KUKA KRL program: sParallel2.src, sParallel2.dat

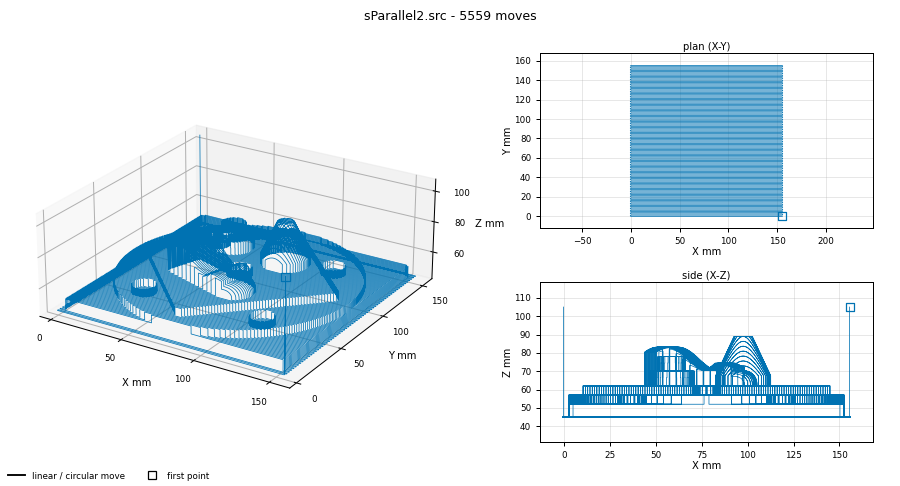
[picture p0: tool path of sParallel2.src, 5559 of 5560 moves have a stored position in this frame; points joined in program order, loops and branches not executed]
--- sParallel2.src ---
&ACCESS RVO
DEF sParallel2()
; Generated by AUTODESK Fusion 360 CAM 2.0.14793
; Creation date: Thursday, March 16, 2023 18:51:27
;FOLD sParallel2
; Start position (joint) = {A1 5,A2 -80,A3 100,A4 75,A5 -60,A6 -65}
; Tool Number            = 4
; Base Number            = 1
; Spindle Speed          = 5000 RPM
; Program file name      = sParallel2.src

PTP {A1 5,A2 -80,A3 100,A4 75,A5 -60,A6 -65,E1 0,E2 0,E3 0,E4 0,E5 0,E6 0}
LIN {X 155.508,Y -0.003,Z 105.000,A 180.000,B 0.000,C 180.000} C_DIS
LIN {X 155.508,Y -0.003,Z 47.000,A 180.000,B 0.000,C 180.000} C_DIS
; Plunge Move Starts
$VEL.CP=0.01
LIN {X 155.508,Y -0.003,Z 45.500,A 180.000,B 0.000,C 180.000} C_DIS
; Lead In Move Starts
LIN {X 155.361,Y -0.003,Z 45.146,A 180.000,B 0.000,C 180.000} C_DIS
LIN {X 155.008,Y -0.003,Z 45.000,A 180.000,B 0.000,C 180.000} C_DIS
; Cutting Move Starts
$VEL.CP=0.02
LIN {X -0.008,Y -0.003,Z 45.000,A 180.000,B 0.000,C 180.000} C_DIS
; Link Move Starts
LIN {X -0.118,Y -0.003,Z 45.026,A 180.000,B 0.000,C 180.000} C_DIS
LIN {X -0.228,Y -0.003,Z 45.051,A 180.000,B 0.000,C 180.000} C_DIS
LIN {X -0.230,Y -0.003,Z 45.051,A 180.000,B 0.000,C 180.000} C_DIS
LIN {X -0.771,Y 0.309,Z 45.051,A 180.000,B 0.000,C 180.000} C_DIS
LIN {X -0.771,Y 0.934,Z 45.051,A 180.000,B 0.000,C 180.000} C_DIS
LIN {X -0.230,Y 1.247,Z 45.051,A 180.000,B 0.000,C 180.000} C_DIS
LIN {X -0.120,Y 1.247,Z 45.026,A 180.000,B 0.000,C 180.000} C_DIS
LIN {X -0.010,Y 1.247,Z 45.000,A 180.000,B 0.000,C 180.000} C_DIS
; Cutting Move Starts
LIN {X 155.010,Y 1.247,Z 45.000,A 180.000,B 0.000,C 180.000} C_DIS
; Link Move Starts
LIN {X 155.120,Y 1.247,Z 45.026,A 180.000,B 0.000,C 180.000} C_DIS
LIN {X 155.230,Y 1.247,Z 45.051,A 180.000,B 0.000,C 180.000} C_DIS
LIN {X 155.771,Y 1.559,Z 45.051,A 180.000,B 0.000,C 180.000} C_DIS
LIN {X 155.771,Y 2.184,Z 45.051,A 180.000,B 0.000,C 180.000} C_DIS
LIN {X 155.230,Y 2.497,Z 45.051,A 180.000,B 0.000,C 180.000} C_DIS
LIN {X 155.120,Y 2.497,Z 45.026,A 180.000,B 0.000,C 180.000} C_DIS
LIN {X 155.010,Y 2.497,Z 45.000,A 180.000,B 0.000,C 180.000} C_DIS
; Cutting Move Starts
LIN {X -0.010,Y 2.497,Z 45.000,A 180.000,B 0.000,C 180.000} C_DIS
; Link Move Starts
LIN {X -0.120,Y 2.497,Z 45.026,A 180.000,B 0.000,C 180.000} C_DIS
LIN {X -0.230,Y 2.497,Z 45.051,A 180.000,B 0.000,C 180.000} C_DIS
LIN {X -0.771,Y 2.809,Z 45.051,A 180.000,B 0.000,C 180.000} C_DIS
LIN {X -0.771,Y 3.434,Z 45.051,A 180.000,B 0.000,C 180.000} C_DIS
LIN {X -0.230,Y 3.746,Z 45.051,A 180.000,B 0.000,C 180.000} C_DIS
LIN {X -0.120,Y 3.746,Z 45.026,A 180.000,B 0.000,C 180.000} C_DIS
LIN {X -0.010,Y 3.746,Z 45.000,A 180.000,B 0.000,C 180.000} C_DIS
; Cutting Move Starts
LIN {X 2.836,Y 3.746,Z 45.000,A 180.000,B 0.000,C 180.000} C_DIS
LIN {X 2.837,Y 3.746,Z 52.000,A 180.000,B 0.000,C 180.000} C_DIS
LIN {X 63.902,Y 3.746,Z 52.000,A 180.000,B 0.000,C 180.000} C_DIS
LIN {X 63.902,Y 3.746,Z 57.000,A 180.000,B 0.000,C 180.000} C_DIS
LIN {X 91.097,Y 3.746,Z 57.000,A 180.000,B 0.000,C 180.000} C_DIS
LIN {X 91.098,Y 3.746,Z 52.000,A 180.000,B 0.000,C 180.000} C_DIS
LIN {X 152.163,Y 3.746,Z 52.000,A 180.000,B 0.000,C 180.000} C_DIS
LIN {X 152.163,Y 3.746,Z 45.000,A 180.000,B 0.000,C 180.000} C_DIS
LIN {X 155.010,Y 3.746,Z 45.000,A 180.000,B 0.000,C 180.000} C_DIS
; Link Move Starts
LIN {X 155.120,Y 3.746,Z 45.026,A 180.000,B 0.000,C 180.000} C_DIS
LIN {X 155.230,Y 3.746,Z 45.051,A 180.000,B 0.000,C 180.000} C_DIS
LIN {X 155.771,Y 4.059,Z 45.051,A 180.000,B 0.000,C 180.000} C_DIS
LIN {X 155.771,Y 4.684,Z 45.051,A 180.000,B 0.000,C 180.000} C_DIS
LIN {X 155.230,Y 4.996,Z 45.051,A 180.000,B 0.000,C 180.000} C_DIS
LIN {X 155.120,Y 4.996,Z 45.026,A 180.000,B 0.000,C 180.000} C_DIS
LIN {X 155.010,Y 4.996,Z 45.000,A 180.000,B 0.000,C 180.000} C_DIS
; Cutting Move Starts
LIN {X 152.500,Y 4.996,Z 45.000,A 180.000,B 0.000,C 180.000} C_DIS
LIN {X 152.500,Y 4.996,Z 52.000,A 180.000,B 0.000,C 180.000} C_DIS
LIN {X 96.687,Y 4.996,Z 52.000,A 180.000,B 0.000,C 180.000} C_DIS
LIN {X 96.684,Y 4.996,Z 57.000,A 180.000,B 0.000,C 180.000} C_DIS
LIN {X 58.313,Y 4.996,Z 57.000,A 180.000,B 0.000,C 180.000} C_DIS
LIN {X 58.313,Y 4.996,Z 52.000,A 180.000,B 0.000,C 180.000} C_DIS
LIN {X 2.500,Y 4.996,Z 52.000,A 180.000,B 0.000,C 180.000} C_DIS
LIN {X 2.500,Y 4.996,Z 45.000,A 180.000,B 0.000,C 180.000} C_DIS
LIN {X -0.010,Y 4.996,Z 45.000,A 180.000,B 0.000,C 180.000} C_DIS
; Link Move Starts
LIN {X -0.120,Y 4.996,Z 45.026,A 180.000,B 0.000,C 180.000} C_DIS
LIN {X -0.230,Y 4.996,Z 45.051,A 180.000,B 0.000,C 180.000} C_DIS
LIN {X -0.771,Y 5.309,Z 45.051,A 180.000,B 0.000,C 180.000} C_DIS
LIN {X -0.771,Y 5.934,Z 45.051,A 180.000,B 0.000,C 180.000} C_DIS
LIN {X -0.230,Y 6.246,Z 45.051,A 180.000,B 0.000,C 180.000} C_DIS
LIN {X -0.120,Y 6.246,Z 45.026,A 180.000,B 0.000,C 180.000} C_DIS
LIN {X -0.010,Y 6.246,Z 45.000,A 180.000,B 0.000,C 180.000} C_DIS
; Cutting Move Starts
LIN {X 2.499,Y 6.246,Z 45.000,A 180.000,B 0.000,C 180.000} C_DIS
LIN {X 2.500,Y 6.246,Z 52.000,A 180.000,B 0.000,C 180.000} C_DIS
LIN {X 54.109,Y 6.246,Z 52.000,A 180.000,B 0.000,C 180.000} C_DIS
LIN {X 54.109,Y 6.246,Z 57.000,A 180.000,B 0.000,C 180.000} C_DIS
LIN {X 100.891,Y 6.246,Z 57.000,A 180.000,B 0.000,C 180.000} C_DIS
LIN {X 100.891,Y 6.246,Z 52.000,A 180.000,B 0.000,C 180.000} C_DIS
LIN {X 152.500,Y 6.246,Z 52.000,A 180.000,B 0.000,C 180.000} C_DIS
LIN {X 152.500,Y 6.246,Z 45.000,A 180.000,B 0.000,C 180.000} C_DIS
LIN {X 155.010,Y 6.246,Z 45.000,A 180.000,B 0.000,C 180.000} C_DIS
; Link Move Starts
LIN {X 155.120,Y 6.246,Z 45.026,A 180.000,B 0.000,C 180.000} C_DIS
LIN {X 155.230,Y 6.246,Z 45.051,A 180.000,B 0.000,C 180.000} C_DIS
LIN {X 155.771,Y 6.559,Z 45.051,A 180.000,B 0.000,C 180.000} C_DIS
LIN {X 155.771,Y 7.184,Z 45.051,A 180.000,B 0.000,C 180.000} C_DIS
LIN {X 155.230,Y 7.496,Z 45.051,A 180.000,B 0.000,C 180.000} C_DIS
LIN {X 155.120,Y 7.496,Z 45.026,A 180.000,B 0.000,C 180.000} C_DIS
LIN {X 155.010,Y 7.496,Z 45.000,A 180.000,B 0.000,C 180.000} C_DIS
; Cutting Move Starts
LIN {X 152.500,Y 7.496,Z 45.000,A 180.000,B 0.000,C 180.000} C_DIS
LIN {X 152.500,Y 7.496,Z 52.000,A 180.000,B 0.000,C 180.000} C_DIS
LIN {X 104.403,Y 7.496,Z 52.000,A 180.000,B 0.000,C 180.000} C_DIS
LIN {X 104.403,Y 7.496,Z 57.000,A 180.000,B 0.000,C 180.000} C_DIS
LIN {X 50.597,Y 7.496,Z 57.000,A 180.000,B 0.000,C 180.000} C_DIS
LIN {X 50.597,Y 7.496,Z 52.000,A 180.000,B 0.000,C 180.000} C_DIS
LIN {X 2.500,Y 7.496,Z 52.000,A 180.000,B 0.000,C 180.000} C_DIS
LIN {X 2.500,Y 7.496,Z 45.000,A 180.000,B 0.000,C 180.000} C_DIS
LIN {X -0.010,Y 7.496,Z 45.000,A 180.000,B 0.000,C 180.000} C_DIS
; Link Move Starts
LIN {X -0.120,Y 7.496,Z 45.026,A 180.000,B 0.000,C 180.000} C_DIS
LIN {X -0.230,Y 7.496,Z 45.051,A 180.000,B 0.000,C 180.000} C_DIS
LIN {X -0.771,Y 7.809,Z 45.051,A 180.000,B 0.000,C 180.000} C_DIS
LIN {X -0.771,Y 8.434,Z 45.051,A 180.000,B 0.000,C 180.000} C_DIS
LIN {X -0.230,Y 8.746,Z 45.051,A 180.000,B 0.000,C 180.000} C_DIS
LIN {X -0.120,Y 8.746,Z 45.026,A 180.000,B 0.000,C 180.000} C_DIS
LIN {X -0.010,Y 8.746,Z 45.000,A 180.000,B 0.000,C 180.000} C_DIS
; Cutting Move Starts
LIN {X 2.500,Y 8.746,Z 45.000,A 180.000,B 0.000,C 180.000} C_DIS
LIN {X 2.500,Y 8.746,Z 52.000,A 180.000,B 0.000,C 180.000} C_DIS
LIN {X 47.548,Y 8.746,Z 52.000,A 180.000,B 0.000,C 180.000} C_DIS
LIN {X 47.548,Y 8.746,Z 57.000,A 180.000,B 0.000,C 180.000} C_DIS
LIN {X 107.452,Y 8.746,Z 57.000,A 180.000,B 0.000,C 180.000} C_DIS
LIN {X 107.452,Y 8.746,Z 52.000,A 180.000,B 0.000,C 180.000} C_DIS
LIN {X 152.500,Y 8.746,Z 52.000,A 180.000,B 0.000,C 180.000} C_DIS
LIN {X 152.500,Y 8.746,Z 45.000,A 180.000,B 0.000,C 180.000} C_DIS
LIN {X 155.010,Y 8.746,Z 45.000,A 180.000,B 0.000,C 180.000} C_DIS
; Link Move Starts
LIN {X 155.120,Y 8.746,Z 45.026,A 180.000,B 0.000,C 180.000} C_DIS
LIN {X 155.230,Y 8.746,Z 45.051,A 180.000,B 0.000,C 180.000} C_DIS
LIN {X 155.771,Y 9.058,Z 45.051,A 180.000,B 0.000,C 180.000} C_DIS
LIN {X 155.771,Y 9.683,Z 45.051,A 180.000,B 0.000,C 180.000} C_DIS
LIN {X 155.230,Y 9.996,Z 45.051,A 180.000,B 0.000,C 180.000} C_DIS
LIN {X 155.120,Y 9.996,Z 45.026,A 180.000,B 0.000,C 180.000} C_DIS
LIN {X 155.010,Y 9.996,Z 45.000,A 180.000,B 0.000,C 180.000} C_DIS
; Cutting Move Starts
LIN {X 152.500,Y 9.996,Z 45.000,A 180.000,B 0.000,C 180.000} C_DIS
LIN {X 152.500,Y 9.996,Z 52.000,A 180.000,B 0.000,C 180.000} C_DIS
LIN {X 110.175,Y 9.996,Z 52.000,A 180.000,B 0.000,C 180.000} C_DIS
LIN {X 110.175,Y 9.996,Z 57.000,A 180.000,B 0.000,C 180.000} C_DIS
LIN {X 44.825,Y 9.996,Z 57.000,A 180.000,B 0.000,C 180.000} C_DIS
LIN {X 44.825,Y 9.996,Z 52.000,A 180.000,B 0.000,C 180.000} C_DIS
LIN {X 2.500,Y 9.996,Z 52.000,A 180.000,B 0.000,C 180.000} C_DIS
LIN {X 2.500,Y 9.996,Z 45.000,A 180.000,B 0.000,C 180.000} C_DIS
LIN {X -0.010,Y 9.996,Z 45.000,A 180.000,B 0.000,C 180.000} C_DIS
; Link Move Starts
LIN {X -0.120,Y 9.996,Z 45.026,A 180.000,B 0.000,C 180.000} C_DIS
LIN {X -0.230,Y 9.996,Z 45.051,A 180.000,B 0.000,C 180.000} C_DIS
LIN {X -0.771,Y 10.308,Z 45.051,A 180.000,B 0.000,C 180.000} C_DIS
LIN {X -0.771,Y 10.933,Z 45.051,A 180.000,B 0.000,C 180.000} C_DIS
LIN {X -0.230,Y 11.246,Z 45.051,A 180.000,B 0.000,C 180.000} C_DIS
LIN {X -0.120,Y 11.246,Z 45.026,A 180.000,B 0.000,C 180.000} C_DIS
LIN {X -0.010,Y 11.246,Z 45.000,A 180.000,B 0.000,C 180.000} C_DIS
; Cutting Move Starts
LIN {X 2.500,Y 11.246,Z 45.000,A 180.000,B 0.000,C 180.000} C_DIS
LIN {X 2.500,Y 11.246,Z 52.000,A 180.000,B 0.000,C 180.000} C_DIS
LIN {X 42.359,Y 11.246,Z 52.000,A 180.000,B 0.000,C 180.000} C_DIS
LIN {X 42.359,Y 11.246,Z 57.000,A 180.000,B 0.000,C 180.000} C_DIS
LIN {X 75.219,Y 11.246,Z 57.000,A 180.000,B 0.000,C 180.000} C_DIS
LIN {X 75.219,Y 11.246,Z 62.000,A 180.000,B 0.000,C 180.000} C_DIS
LIN {X 79.781,Y 11.246,Z 62.000,A 180.000,B 0.000,C 180.000} C_DIS
LIN {X 79.781,Y 11.246,Z 57.000,A 180.000,B 0.000,C 180.000} C_DIS
LIN {X 112.641,Y 11.246,Z 57.000,A 180.000,B 0.000,C 180.000} C_DIS
LIN {X 112.641,Y 11.246,Z 52.000,A 180.000,B 0.000,C 180.000} C_DIS
LIN {X 152.500,Y 11.246,Z 52.000,A 180.000,B 0.000,C 180.000} C_DIS
LIN {X 152.500,Y 11.246,Z 45.000,A 180.000,B 0.000,C 180.000} C_DIS
LIN {X 155.010,Y 11.246,Z 45.000,A 180.000,B 0.000,C 180.000} C_DIS
; Link Move Starts
LIN {X 155.120,Y 11.246,Z 45.026,A 180.000,B 0.000,C 180.000} C_DIS
LIN {X 155.230,Y 11.246,Z 45.051,A 180.000,B 0.000,C 180.000} C_DIS
LIN {X 155.771,Y 11.558,Z 45.051,A 180.000,B 0.000,C 180.000} C_DIS
LIN {X 155.771,Y 12.183,Z 45.051,A 180.000,B 0.000,C 180.000} C_DIS
LIN {X 155.230,Y 12.496,Z 45.051,A 180.000,B 0.000,C 180.000} C_DIS
LIN {X 155.120,Y 12.496,Z 45.026,A 180.000,B 0.000,C 180.000} C_DIS
LIN {X 155.010,Y 12.496,Z 45.000,A 180.000,B 0.000,C 180.000} C_DIS
; Cutting Move Starts
LIN {X 152.500,Y 12.496,Z 45.000,A 180.000,B 0.000,C 180.000} C_DIS
LIN {X 152.500,Y 12.496,Z 52.000,A 180.000,B 0.000,C 180.000} C_DIS
LIN {X 114.901,Y 12.496,Z 52.000,A 180.000,B 0.000,C 180.000} C_DIS
LIN {X 114.901,Y 12.496,Z 57.000,A 180.000,B 0.000,C 180.000} C_DIS
LIN {X 81.031,Y 12.496,Z 57.000,A 180.000,B 0.000,C 180.000} C_DIS
LIN {X 81.031,Y 12.496,Z 62.000,A 180.000,B 0.000,C 180.000} C_DIS
LIN {X 73.969,Y 12.496,Z 62.000,A 180.000,B 0.000,C 180.000} C_DIS
LIN {X 73.969,Y 12.496,Z 57.000,A 180.000,B 0.000,C 180.000} C_DIS
LIN {X 40.099,Y 12.496,Z 57.000,A 180.000,B 0.000,C 180.000} C_DIS
LIN {X 40.099,Y 12.496,Z 52.000,A 180.000,B 0.000,C 180.000} C_DIS
LIN {X 2.500,Y 12.496,Z 52.000,A 180.000,B 0.000,C 180.000} C_DIS
LIN {X 2.500,Y 12.496,Z 45.000,A 180.000,B 0.000,C 180.000} C_DIS
LIN {X -0.010,Y 12.496,Z 45.000,A 180.000,B 0.000,C 180.000} C_DIS
; Link Move Starts
LIN {X -0.120,Y 12.496,Z 45.026,A 180.000,B 0.000,C 180.000} C_DIS
LIN {X -0.230,Y 12.496,Z 45.051,A 180.000,B 0.000,C 180.000} C_DIS
LIN {X -0.771,Y 12.808,Z 45.051,A 180.000,B 0.000,C 180.000} C_DIS
LIN {X -0.771,Y 13.433,Z 45.051,A 180.000,B 0.000,C 180.000} C_DIS
LIN {X -0.230,Y 13.746,Z 45.051,A 180.000,B 0.000,C 180.000} C_DIS
LIN {X -0.120,Y 13.746,Z 45.026,A 180.000,B 0.000,C 180.000} C_DIS
LIN {X -0.010,Y 13.746,Z 45.000,A 180.000,B 0.000,C 180.000} C_DIS
; Cutting Move Starts
LIN {X 2.498,Y 13.746,Z 45.000,A 180.000,B 0.000,C 180.000} C_DIS
LIN {X 2.500,Y 13.746,Z 52.000,A 180.000,B 0.000,C 180.000} C_DIS
LIN {X 38.007,Y 13.746,Z 52.000,A 180.000,B 0.000,C 180.000} C_DIS
LIN {X 38.007,Y 13.746,Z 57.000,A 180.000,B 0.000,C 180.000} C_DIS
LIN {X 72.716,Y 13.746,Z 57.000,A 180.000,B 0.000,C 180.000} C_DIS
LIN {X 72.719,Y 13.746,Z 62.000,A 180.000,B 0.000,C 180.000} C_DIS
LIN {X 82.281,Y 13.746,Z 62.000,A 180.000,B 0.000,C 180.000} C_DIS
LIN {X 82.281,Y 13.746,Z 57.000,A 180.000,B 0.000,C 180.000} C_DIS
LIN {X 116.993,Y 13.746,Z 57.000,A 180.000,B 0.000,C 180.000} C_DIS
LIN {X 116.993,Y 13.746,Z 52.000,A 180.000,B 0.000,C 180.000} C_DIS
LIN {X 152.500,Y 13.746,Z 52.000,A 180.000,B 0.000,C 180.000} C_DIS
LIN {X 152.500,Y 13.746,Z 45.000,A 180.000,B 0.000,C 180.000} C_DIS
LIN {X 155.010,Y 13.746,Z 45.000,A 180.000,B 0.000,C 180.000} C_DIS
; Link Move Starts
LIN {X 155.120,Y 13.746,Z 45.026,A 180.000,B 0.000,C 180.000} C_DIS
LIN {X 155.230,Y 13.746,Z 45.051,A 180.000,B 0.000,C 180.000} C_DIS
LIN {X 155.771,Y 14.058,Z 45.051,A 180.000,B 0.000,C 180.000} C_DIS
LIN {X 155.771,Y 14.683,Z 45.051,A 180.000,B 0.000,C 180.000} C_DIS
LIN {X 155.230,Y 14.996,Z 45.051,A 180.000,B 0.000,C 180.000} C_DIS
LIN {X 155.120,Y 14.996,Z 45.026,A 180.000,B 0.000,C 180.000} C_DIS
LIN {X 155.010,Y 14.996,Z 45.000,A 180.000,B 0.000,C 180.000} C_DIS
; Cutting Move Starts
LIN {X 152.500,Y 14.996,Z 45.000,A 180.000,B 0.000,C 180.000} C_DIS
LIN {X 152.500,Y 14.996,Z 52.000,A 180.000,B 0.000,C 180.000} C_DIS
LIN {X 118.951,Y 14.996,Z 52.000,A 180.000,B 0.000,C 180.000} C_DIS
LIN {X 118.950,Y 14.996,Z 57.000,A 180.000,B 0.000,C 180.000} C_DIS
LIN {X 83.531,Y 14.996,Z 57.000,A 180.000,B 0.000,C 180.000} C_DIS
LIN {X 83.531,Y 14.996,Z 62.000,A 180.000,B 0.000,C 180.000} C_DIS
LIN {X 71.469,Y 14.996,Z 62.000,A 180.000,B 0.000,C 180.000} C_DIS
LIN {X 71.469,Y 14.996,Z 57.000,A 180.000,B 0.000,C 180.000} C_DIS
LIN {X 36.049,Y 14.996,Z 57.000,A 180.000,B 0.000,C 180.000} C_DIS
LIN {X 36.049,Y 14.996,Z 52.000,A 180.000,B 0.000,C 180.000} C_DIS
LIN {X 2.500,Y 14.996,Z 52.000,A 180.000,B 0.000,C 180.000} C_DIS
LIN {X 2.499,Y 14.996,Z 45.000,A 180.000,B 0.000,C 180.000} C_DIS
LIN {X -0.010,Y 14.996,Z 45.000,A 180.000,B 0.000,C 180.000} C_DIS
; Link Move Starts
LIN {X -0.120,Y 14.996,Z 45.026,A 180.000,B 0.000,C 180.000} C_DIS
LIN {X -0.230,Y 14.996,Z 45.051,A 180.000,B 0.000,C 180.000} C_DIS
LIN {X -0.771,Y 15.308,Z 45.051,A 180.000,B 0.000,C 180.000} C_DIS
LIN {X -0.771,Y 15.933,Z 45.051,A 180.000,B 0.000,C 180.000} C_DIS
LIN {X -0.230,Y 16.245,Z 45.051,A 180.000,B 0.000,C 180.000} C_DIS
LIN {X -0.120,Y 16.245,Z 45.026,A 180.000,B 0.000,C 180.000} C_DIS
LIN {X -0.010,Y 16.245,Z 45.000,A 180.000,B 0.000,C 180.000} C_DIS
; Cutting Move Starts
LIN {X 2.500,Y 16.245,Z 45.000,A 180.000,B 0.000,C 180.000} C_DIS
LIN {X 2.500,Y 16.245,Z 52.000,A 180.000,B 0.000,C 180.000} C_DIS
LIN {X 34.229,Y 16.245,Z 52.000,A 180.000,B 0.000,C 180.000} C_DIS
LIN {X 34.229,Y 16.245,Z 57.000,A 180.000,B 0.000,C 180.000} C_DIS
LIN {X 70.219,Y 16.245,Z 57.000,A 180.000,B 0.000,C 180.000} C_DIS
LIN {X 70.219,Y 16.245,Z 62.000,A 180.000,B 0.000,C 180.000} C_DIS
LIN {X 84.781,Y 16.245,Z 62.000,A 180.000,B 0.000,C 180.000} C_DIS
LIN {X 84.781,Y 16.245,Z 57.000,A 180.000,B 0.000,C 180.000} C_DIS
LIN {X 120.771,Y 16.245,Z 57.000,A 180.000,B 0.000,C 180.000} C_DIS
LIN {X 120.771,Y 16.245,Z 52.000,A 180.000,B 0.000,C 180.000} C_DIS
LIN {X 152.500,Y 16.245,Z 52.000,A 180.000,B 0.000,C 180.000} C_DIS
LIN {X 152.500,Y 16.245,Z 45.000,A 180.000,B 0.000,C 180.000} C_DIS
LIN {X 155.010,Y 16.245,Z 45.000,A 180.000,B 0.000,C 180.000} C_DIS
; Link Move Starts
LIN {X 155.120,Y 16.245,Z 45.026,A 180.000,B 0.000,C 180.000} C_DIS
LIN {X 155.230,Y 16.245,Z 45.051,A 180.000,B 0.000,C 180.000} C_DIS
LIN {X 155.771,Y 16.558,Z 45.051,A 180.000,B 0.000,C 180.000} C_DIS
LIN {X 155.771,Y 17.183,Z 45.051,A 180.000,B 0.000,C 180.000} C_DIS
LIN {X 155.230,Y 17.495,Z 45.051,A 180.000,B 0.000,C 180.000} C_DIS
LIN {X 155.120,Y 17.495,Z 45.026,A 180.000,B 0.000,C 180.000} C_DIS
LIN {X 155.010,Y 17.495,Z 45.000,A 180.000,B 0.000,C 180.000} C_DIS
; Cutting Move Starts
LIN {X 152.500,Y 17.495,Z 45.000,A 180.000,B 0.000,C 180.000} C_DIS
LIN {X 152.500,Y 17.495,Z 52.000,A 180.000,B 0.000,C 180.000} C_DIS
LIN {X 122.486,Y 17.495,Z 52.000,A 180.000,B 0.000,C 180.000} C_DIS
LIN {X 122.486,Y 17.495,Z 57.000,A 180.000,B 0.000,C 180.000} C_DIS
LIN {X 86.031,Y 17.495,Z 57.000,A 180.000,B 0.000,C 180.000} C_DIS
LIN {X 86.030,Y 17.495,Z 62.000,A 180.000,B 0.000,C 180.000} C_DIS
LIN {X 68.969,Y 17.495,Z 62.000,A 180.000,B 0.000,C 180.000} C_DIS
LIN {X 68.969,Y 17.495,Z 57.000,A 180.000,B 0.000,C 180.000} C_DIS
LIN {X 32.514,Y 17.495,Z 57.000,A 180.000,B 0.000,C 180.000} C_DIS
LIN {X 32.512,Y 17.495,Z 52.000,A 180.000,B 0.000,C 180.000} C_DIS
LIN {X 2.500,Y 17.495,Z 52.000,A 180.000,B 0.000,C 180.000} C_DIS
LIN {X 2.500,Y 17.495,Z 45.000,A 180.000,B 0.000,C 180.000} C_DIS
LIN {X -0.010,Y 17.495,Z 45.000,A 180.000,B 0.000,C 180.000} C_DIS
; Link Move Starts
LIN {X -0.120,Y 17.495,Z 45.026,A 180.000,B 0.000,C 180.000} C_DIS
LIN {X -0.230,Y 17.495,Z 45.051,A 180.000,B 0.000,C 180.000} C_DIS
LIN {X -0.771,Y 17.808,Z 45.051,A 180.000,B 0.000,C 180.000} C_DIS
LIN {X -0.771,Y 18.433,Z 45.051,A 180.000,B 0.000,C 180.000} C_DIS
LIN {X -0.230,Y 18.745,Z 45.051,A 180.000,B 0.000,C 180.000} C_DIS
LIN {X -0.120,Y 18.745,Z 45.026,A 180.000,B 0.000,C 180.000} C_DIS
LIN {X -0.010,Y 18.745,Z 45.000,A 180.000,B 0.000,C 180.000} C_DIS
; Cutting Move Starts
LIN {X 2.500,Y 18.745,Z 45.000,A 180.000,B 0.000,C 180.000} C_DIS
LIN {X 2.500,Y 18.745,Z 52.000,A 180.000,B 0.000,C 180.000} C_DIS
LIN {X 30.894,Y 18.745,Z 52.000,A 180.000,B 0.000,C 180.000} C_DIS
LIN {X 30.894,Y 18.745,Z 57.000,A 180.000,B 0.000,C 180.000} C_DIS
LIN {X 67.719,Y 18.745,Z 57.000,A 180.000,B 0.000,C 180.000} C_DIS
LIN {X 67.719,Y 18.745,Z 62.000,A 180.000,B 0.000,C 180.000} C_DIS
LIN {X 87.281,Y 18.745,Z 62.000,A 180.000,B 0.000,C 180.000} C_DIS
LIN {X 87.281,Y 18.745,Z 57.000,A 180.000,B 0.000,C 180.000} C_DIS
LIN {X 124.106,Y 18.745,Z 57.000,A 180.000,B 0.000,C 180.000} C_DIS
LIN {X 124.106,Y 18.745,Z 52.000,A 180.000,B 0.000,C 180.000} C_DIS
LIN {X 152.500,Y 18.745,Z 52.000,A 180.000,B 0.000,C 180.000} C_DIS
LIN {X 152.500,Y 18.745,Z 45.000,A 180.000,B 0.000,C 180.000} C_DIS
LIN {X 155.010,Y 18.745,Z 45.000,A 180.000,B 0.000,C 180.000} C_DIS
; Link Move Starts
LIN {X 155.120,Y 18.745,Z 45.026,A 180.000,B 0.000,C 180.000} C_DIS
LIN {X 155.230,Y 18.745,Z 45.051,A 180.000,B 0.000,C 180.000} C_DIS
LIN {X 155.771,Y 19.058,Z 45.051,A 180.000,B 0.000,C 180.000} C_DIS
LIN {X 155.771,Y 19.683,Z 45.051,A 180.000,B 0.000,C 180.000} C_DIS
LIN {X 155.230,Y 19.995,Z 45.051,A 180.000,B 0.000,C 180.000} C_DIS
LIN {X 155.120,Y 19.995,Z 45.026,A 180.000,B 0.000,C 180.000} C_DIS
LIN {X 155.010,Y 19.995,Z 45.000,A 180.000,B 0.000,C 180.000} C_DIS
; Cutting Move Starts
LIN {X 152.500,Y 19.995,Z 45.000,A 180.000,B 0.000,C 180.000} C_DIS
LIN {X 152.500,Y 19.995,Z 52.000,A 180.000,B 0.000,C 180.000} C_DIS
LIN {X 125.641,Y 19.995,Z 52.000,A 180.000,B 0.000,C 180.000} C_DIS
LIN {X 125.640,Y 19.995,Z 57.000,A 180.000,B 0.000,C 180.000} C_DIS
LIN {X 88.531,Y 19.995,Z 57.000,A 180.000,B 0.000,C 180.000} C_DIS
LIN {X 88.528,Y 19.995,Z 62.000,A 180.000,B 0.000,C 180.000} C_DIS
LIN {X 66.469,Y 19.995,Z 62.000,A 180.000,B 0.000,C 180.000} C_DIS
LIN {X 66.469,Y 19.995,Z 57.000,A 180.000,B 0.000,C 180.000} C_DIS
LIN {X 29.359,Y 19.995,Z 57.000,A 180.000,B 0.000,C 180.000} C_DIS
LIN {X 29.355,Y 19.995,Z 52.000,A 180.000,B 0.000,C 180.000} C_DIS
LIN {X 2.500,Y 19.995,Z 52.000,A 180.000,B 0.000,C 180.000} C_DIS
LIN {X 2.500,Y 19.995,Z 45.000,A 180.000,B 0.000,C 180.000} C_DIS
LIN {X -0.010,Y 19.995,Z 45.000,A 180.000,B 0.000,C 180.000} C_DIS
; Link Move Starts
LIN {X -0.120,Y 19.995,Z 45.026,A 180.000,B 0.000,C 180.000} C_DIS
LIN {X -0.230,Y 19.995,Z 45.051,A 180.000,B 0.000,C 180.000} C_DIS
LIN {X -0.771,Y 20.308,Z 45.051,A 180.000,B 0.000,C 180.000} C_DIS
LIN {X -0.771,Y 20.933,Z 45.051,A 180.000,B 0.000,C 180.000} C_DIS
LIN {X -0.230,Y 21.245,Z 45.051,A 180.000,B 0.000,C 180.000} C_DIS
LIN {X -0.120,Y 21.245,Z 45.026,A 180.000,B 0.000,C 180.000} C_DIS
LIN {X -0.010,Y 21.245,Z 45.000,A 180.000,B 0.000,C 180.000} C_DIS
; Cutting Move Starts
LIN {X 2.496,Y 21.245,Z 45.000,A 180.000,B 0.000,C 180.000} C_DIS
LIN {X 2.500,Y 21.245,Z 52.000,A 180.000,B 0.000,C 180.000} C_DIS
LIN {X 27.902,Y 21.245,Z 52.000,A 180.000,B 0.000,C 180.000} C_DIS
LIN {X 27.902,Y 21.245,Z 57.000,A 180.000,B 0.000,C 180.000} C_DIS
LIN {X 65.216,Y 21.245,Z 57.000,A 180.000,B 0.000,C 180.000} C_DIS
LIN {X 65.219,Y 21.245,Z 62.000,A 180.000,B 0.000,C 180.000} C_DIS
LIN {X 89.781,Y 21.245,Z 62.000,A 180.000,B 0.000,C 180.000} C_DIS
LIN {X 89.781,Y 21.245,Z 57.000,A 180.000,B 0.000,C 180.000} C_DIS
LIN {X 127.094,Y 21.245,Z 57.000,A 180.000,B 0.000,C 180.000} C_DIS
LIN {X 127.098,Y 21.245,Z 52.000,A 180.000,B 0.000,C 180.000} C_DIS
LIN {X 152.500,Y 21.245,Z 52.000,A 180.000,B 0.000,C 180.000} C_DIS
LIN {X 152.500,Y 21.245,Z 45.000,A 180.000,B 0.000,C 180.000} C_DIS
LIN {X 155.010,Y 21.245,Z 45.000,A 180.000,B 0.000,C 180.000} C_DIS
; Link Move Starts
LIN {X 155.120,Y 21.245,Z 45.026,A 180.000,B 0.000,C 180.000} C_DIS
LIN {X 155.230,Y 21.245,Z 45.051,A 180.000,B 0.000,C 180.000} C_DIS
LIN {X 155.771,Y 21.557,Z 45.051,A 180.000,B 0.000,C 180.000} C_DIS
LIN {X 155.771,Y 22.182,Z 45.051,A 180.000,B 0.000,C 180.000} C_DIS
LIN {X 155.230,Y 22.495,Z 45.051,A 180.000,B 0.000,C 180.000} C_DIS
LIN {X 155.120,Y 22.495,Z 45.026,A 180.000,B 0.000,C 180.000} C_DIS
LIN {X 155.010,Y 22.495,Z 45.000,A 180.000,B 0.000,C 180.000} C_DIS
; Cutting Move Starts
LIN {X 152.500,Y 22.495,Z 45.000,A 180.000,B 0.000,C 180.000} C_DIS
LIN {X 152.500,Y 22.495,Z 52.000,A 180.000,B 0.000,C 180.000} C_DIS
LIN {X 128.482,Y 22.495,Z 52.000,A 180.000,B 0.000,C 180.000} C_DIS
LIN {X 128.482,Y 22.495,Z 57.000,A 180.000,B 0.000,C 180.000} C_DIS
LIN {X 91.030,Y 22.495,Z 57.000,A 180.000,B 0.000,C 180.000} C_DIS
LIN {X 91.030,Y 22.495,Z 62.000,A 180.000,B 0.000,C 180.000} C_DIS
LIN {X 63.970,Y 22.495,Z 62.000,A 180.000,B 0.000,C 180.000} C_DIS
LIN {X 63.970,Y 22.495,Z 57.000,A 180.000,B 0.000,C 180.000} C_DIS
LIN {X 26.518,Y 22.495,Z 57.000,A 180.000,B 0.000,C 180.000} C_DIS
LIN {X 26.518,Y 22.495,Z 52.000,A 180.000,B 0.000,C 180.000} C_DIS
LIN {X 2.500,Y 22.495,Z 52.000,A 180.000,B 0.000,C 180.000} C_DIS
LIN {X 2.500,Y 22.495,Z 45.000,A 180.000,B 0.000,C 180.000} C_DIS
LIN {X -0.010,Y 22.495,Z 45.000,A 180.000,B 0.000,C 180.000} C_DIS
; Link Move Starts
LIN {X -0.120,Y 22.495,Z 45.026,A 180.000,B 0.000,C 180.000} C_DIS
LIN {X -0.230,Y 22.495,Z 45.051,A 180.000,B 0.000,C 180.000} C_DIS
LIN {X -0.771,Y 22.807,Z 45.051,A 180.000,B 0.000,C 180.000} C_DIS
LIN {X -0.771,Y 23.432,Z 45.051,A 180.000,B 0.000,C 180.000} C_DIS
LIN {X -0.230,Y 23.745,Z 45.051,A 180.000,B 0.000,C 180.000} C_DIS
LIN {X -0.120,Y 23.745,Z 45.026,A 180.000,B 0.000,C 180.000} C_DIS
LIN {X -0.010,Y 23.745,Z 45.000,A 180.000,B 0.000,C 180.000} C_DIS
; Cutting Move Starts
LIN {X 2.500,Y 23.745,Z 45.000,A 180.000,B 0.000,C 180.000} C_DIS
LIN {X 2.500,Y 23.745,Z 52.000,A 180.000,B 0.000,C 180.000} C_DIS
LIN {X 25.201,Y 23.745,Z 52.000,A 180.000,B 0.000,C 180.000} C_DIS
LIN {X 25.201,Y 23.745,Z 57.000,A 180.000,B 0.000,C 180.000} C_DIS
LIN {X 62.720,Y 23.745,Z 57.000,A 180.000,B 0.000,C 180.000} C_DIS
LIN {X 62.720,Y 23.745,Z 62.000,A 180.000,B 0.000,C 180.000} C_DIS
LIN {X 92.280,Y 23.745,Z 62.000,A 180.000,B 0.000,C 180.000} C_DIS
LIN {X 92.280,Y 23.745,Z 57.000,A 180.000,B 0.000,C 180.000} C_DIS
LIN {X 129.799,Y 23.745,Z 57.000,A 180.000,B 0.000,C 180.000} C_DIS
LIN {X 129.799,Y 23.745,Z 52.000,A 180.000,B 0.000,C 180.000} C_DIS
LIN {X 152.500,Y 23.745,Z 52.000,A 180.000,B 0.000,C 180.000} C_DIS
LIN {X 152.500,Y 23.745,Z 45.000,A 180.000,B 0.000,C 180.000} C_DIS
LIN {X 155.010,Y 23.745,Z 45.000,A 180.000,B 0.000,C 180.000} C_DIS
; Link Move Starts
LIN {X 155.120,Y 23.745,Z 45.026,A 180.000,B 0.000,C 180.000} C_DIS
LIN {X 155.230,Y 23.745,Z 45.051,A 180.000,B 0.000,C 180.000} C_DIS
LIN {X 155.771,Y 24.057,Z 45.051,A 180.000,B 0.000,C 180.000} C_DIS
LIN {X 155.771,Y 24.682,Z 45.051,A 180.000,B 0.000,C 180.000} C_DIS
LIN {X 155.230,Y 24.995,Z 45.051,A 180.000,B 0.000,C 180.000} C_DIS
LIN {X 155.120,Y 24.995,Z 45.026,A 180.000,B 0.000,C 180.000} C_DIS
LIN {X 155.010,Y 24.995,Z 45.000,A 180.000,B 0.000,C 180.000} C_DIS
; Cutting Move Starts
LIN {X 152.500,Y 24.995,Z 45.000,A 180.000,B 0.000,C 180.000} C_DIS
LIN {X 152.500,Y 24.995,Z 52.000,A 180.000,B 0.000,C 180.000} C_DIS
LIN {X 131.054,Y 24.995,Z 52.000,A 180.000,B 0.000,C 180.000} C_DIS
LIN {X 131.054,Y 24.995,Z 57.000,A 180.000,B 0.000,C 180.000} C_DIS
LIN {X 93.530,Y 24.995,Z 57.000,A 180.000,B 0.000,C 180.000} C_DIS
LIN {X 93.527,Y 24.995,Z 62.000,A 180.000,B 0.000,C 180.000} C_DIS
LIN {X 61.470,Y 24.995,Z 62.000,A 180.000,B 0.000,C 180.000} C_DIS
LIN {X 61.470,Y 24.995,Z 57.000,A 180.000,B 0.000,C 180.000} C_DIS
LIN {X 23.946,Y 24.995,Z 57.000,A 180.000,B 0.000,C 180.000} C_DIS
LIN {X 23.946,Y 24.995,Z 52.000,A 180.000,B 0.000,C 180.000} C_DIS
LIN {X 2.500,Y 24.995,Z 52.000,A 180.000,B 0.000,C 180.000} C_DIS
LIN {X 2.500,Y 24.995,Z 45.000,A 180.000,B 0.000,C 180.000} C_DIS
LIN {X -0.010,Y 24.995,Z 45.000,A 180.000,B 0.000,C 180.000} C_DIS
; Link Move Starts
LIN {X -0.120,Y 24.995,Z 45.026,A 180.000,B 0.000,C 180.000} C_DIS
LIN {X -0.230,Y 24.995,Z 45.051,A 180.000,B 0.000,C 180.000} C_DIS
LIN {X -0.771,Y 25.307,Z 45.051,A 180.000,B 0.000,C 180.000} C_DIS
LIN {X -0.771,Y 25.932,Z 45.051,A 180.000,B 0.000,C 180.000} C_DIS
LIN {X -0.230,Y 26.245,Z 45.051,A 180.000,B 0.000,C 180.000} C_DIS
LIN {X -0.120,Y 26.245,Z 45.026,A 180.000,B 0.000,C 180.000} C_DIS
LIN {X -0.010,Y 26.245,Z 45.000,A 180.000,B 0.000,C 180.000} C_DIS
; Cutting Move Starts
LIN {X 2.500,Y 26.245,Z 45.000,A 180.000,B 0.000,C 180.000} C_DIS
LIN {X 2.500,Y 26.245,Z 52.000,A 180.000,B 0.000,C 180.000} C_DIS
LIN {X 22.749,Y 26.245,Z 52.000,A 180.000,B 0.000,C 180.000} C_DIS
LIN {X 22.749,Y 26.245,Z 57.000,A 180.000,B 0.000,C 180.000} C_DIS
LIN {X 60.220,Y 26.245,Z 57.000,A 180.000,B 0.000,C 180.000} C_DIS
LIN {X 60.220,Y 26.245,Z 62.000,A 180.000,B 0.000,C 180.000} C_DIS
LIN {X 94.780,Y 26.245,Z 62.000,A 180.000,B 0.000,C 180.000} C_DIS
LIN {X 94.780,Y 26.245,Z 57.000,A 180.000,B 0.000,C 180.000} C_DIS
LIN {X 132.251,Y 26.245,Z 57.000,A 180.000,B 0.000,C 180.000} C_DIS
LIN {X 132.251,Y 26.245,Z 52.000,A 180.000,B 0.000,C 180.000} C_DIS
LIN {X 152.500,Y 26.245,Z 52.000,A 180.000,B 0.000,C 180.000} C_DIS
LIN {X 152.500,Y 26.245,Z 45.000,A 180.000,B 0.000,C 180.000} C_DIS
LIN {X 155.010,Y 26.245,Z 45.000,A 180.000,B 0.000,C 180.000} C_DIS
; Link Move Starts
LIN {X 155.120,Y 26.245,Z 45.026,A 180.000,B 0.000,C 180.000} C_DIS
LIN {X 155.230,Y 26.245,Z 45.051,A 180.000,B 0.000,C 180.000} C_DIS
LIN {X 155.771,Y 26.557,Z 45.051,A 180.000,B 0.000,C 180.000} C_DIS
LIN {X 155.771,Y 27.182,Z 45.051,A 180.000,B 0.000,C 180.000} C_DIS
LIN {X 155.230,Y 27.495,Z 45.051,A 180.000,B 0.000,C 180.000} C_DIS
LIN {X 155.120,Y 27.495,Z 45.026,A 180.000,B 0.000,C 180.000} C_DIS
LIN {X 155.010,Y 27.495,Z 45.000,A 180.000,B 0.000,C 180.000} C_DIS
; Cutting Move Starts
LIN {X 152.500,Y 27.495,Z 45.000,A 180.000,B 0.000,C 180.000} C_DIS
LIN {X 152.500,Y 27.495,Z 52.000,A 180.000,B 0.000,C 180.000} C_DIS
LIN {X 133.394,Y 27.495,Z 52.000,A 180.000,B 0.000,C 180.000} C_DIS
LIN {X 133.394,Y 27.495,Z 57.000,A 180.000,B 0.000,C 180.000} C_DIS
LIN {X 96.030,Y 27.495,Z 57.000,A 180.000,B 0.000,C 180.000} C_DIS
LIN {X 96.030,Y 27.495,Z 62.000,A 180.000,B 0.000,C 180.000} C_DIS
LIN {X 58.970,Y 27.495,Z 62.000,A 180.000,B 0.000,C 180.000} C_DIS
LIN {X 58.970,Y 27.495,Z 57.000,A 180.000,B 0.000,C 180.000} C_DIS
LIN {X 21.606,Y 27.495,Z 57.000,A 180.000,B 0.000,C 180.000} C_DIS
LIN {X 21.606,Y 27.495,Z 52.000,A 180.000,B 0.000,C 180.000} C_DIS
LIN {X 2.500,Y 27.495,Z 52.000,A 180.000,B 0.000,C 180.000} C_DIS
LIN {X 2.500,Y 27.495,Z 45.000,A 180.000,B 0.000,C 180.000} C_DIS
LIN {X -0.010,Y 27.495,Z 45.000,A 180.000,B 0.000,C 180.000} C_DIS
; Link Move Starts
LIN {X -0.120,Y 27.495,Z 45.026,A 180.000,B 0.000,C 180.000} C_DIS
LIN {X -0.230,Y 27.495,Z 45.051,A 180.000,B 0.000,C 180.000} C_DIS
LIN {X -0.771,Y 27.807,Z 45.051,A 180.000,B 0.000,C 180.000} C_DIS
LIN {X -0.771,Y 28.432,Z 45.051,A 180.000,B 0.000,C 180.000} C_DIS
LIN {X -0.230,Y 28.744,Z 45.051,A 180.000,B 0.000,C 180.000} C_DIS
LIN {X -0.120,Y 28.744,Z 45.026,A 180.000,B 0.000,C 180.000} C_DIS
LIN {X -0.010,Y 28.744,Z 45.000,A 180.000,B 0.000,C 180.000} C_DIS
; Cutting Move Starts
LIN {X 2.500,Y 28.744,Z 45.000,A 180.000,B 0.000,C 180.000} C_DIS
LIN {X 2.500,Y 28.744,Z 52.000,A 180.000,B 0.000,C 180.000} C_DIS
LIN {X 20.514,Y 28.744,Z 52.000,A 180.000,B 0.000,C 180.000} C_DIS
LIN {X 20.514,Y 28.744,Z 57.000,A 180.000,B 0.000,C 180.000} C_DIS
LIN {X 57.717,Y 28.744,Z 57.000,A 180.000,B 0.000,C 180.000} C_DIS
LIN {X 57.720,Y 28.744,Z 62.000,A 180.000,B 0.000,C 180.000} C_DIS
LIN {X 97.280,Y 28.744,Z 62.000,A 180.000,B 0.000,C 180.000} C_DIS
LIN {X 97.280,Y 28.744,Z 57.000,A 180.000,B 0.000,C 180.000} C_DIS
LIN {X 134.486,Y 28.744,Z 57.000,A 180.000,B 0.000,C 180.000} C_DIS
LIN {X 134.486,Y 28.744,Z 52.000,A 180.000,B 0.000,C 180.000} C_DIS
LIN {X 152.500,Y 28.744,Z 52.000,A 180.000,B 0.000,C 180.000} C_DIS
LIN {X 152.500,Y 28.744,Z 45.000,A 180.000,B 0.000,C 180.000} C_DIS
LIN {X 155.010,Y 28.744,Z 45.000,A 180.000,B 0.000,C 180.000} C_DIS
; Link Move Starts
LIN {X 155.120,Y 28.744,Z 45.026,A 180.000,B 0.000,C 180.000} C_DIS
LIN {X 155.230,Y 28.744,Z 45.051,A 180.000,B 0.000,C 180.000} C_DIS
LIN {X 155.771,Y 29.057,Z 45.051,A 180.000,B 0.000,C 180.000} C_DIS
LIN {X 155.771,Y 29.682,Z 45.051,A 180.000,B 0.000,C 180.000} C_DIS
LIN {X 155.230,Y 29.994,Z 45.051,A 180.000,B 0.000,C 180.000} C_DIS
LIN {X 155.120,Y 29.994,Z 45.026,A 180.000,B 0.000,C 180.000} C_DIS
LIN {X 155.010,Y 29.994,Z 45.000,A 180.000,B 0.000,C 180.000} C_DIS
; Cutting Move Starts
LIN {X 152.500,Y 29.994,Z 45.000,A 180.000,B 0.000,C 180.000} C_DIS
LIN {X 152.500,Y 29.994,Z 52.000,A 180.000,B 0.000,C 180.000} C_DIS
LIN {X 135.531,Y 29.994,Z 52.000,A 180.000,B 0.000,C 180.000} C_DIS
LIN {X 135.527,Y 29.994,Z 57.000,A 180.000,B 0.000,C 180.000} C_DIS
LIN {X 122.223,Y 29.994,Z 57.000,A 180.000,B 0.000,C 180.000} C_DIS
LIN {X 122.223,Y 29.994,Z 52.000,A 180.000,B 0.000,C 180.000} C_DIS
LIN {X 114.777,Y 29.994,Z 52.000,A 180.000,B 0.000,C 180.000} C_DIS
LIN {X 114.777,Y 29.994,Z 57.000,A 180.000,B 0.000,C 180.000} C_DIS
LIN {X 98.530,Y 29.994,Z 57.000,A 180.000,B 0.000,C 180.000} C_DIS
LIN {X 98.530,Y 29.994,Z 62.000,A 180.000,B 0.000,C 180.000} C_DIS
LIN {X 56.470,Y 29.994,Z 62.000,A 180.000,B 0.000,C 180.000} C_DIS
LIN {X 56.470,Y 29.994,Z 57.000,A 180.000,B 0.000,C 180.000} C_DIS
LIN {X 40.223,Y 29.994,Z 57.000,A 180.000,B 0.000,C 180.000} C_DIS
LIN {X 40.223,Y 29.994,Z 52.000,A 180.000,B 0.000,C 180.000} C_DIS
LIN {X 32.777,Y 29.994,Z 52.000,A 180.000,B 0.000,C 180.000} C_DIS
LIN {X 32.777,Y 29.994,Z 57.000,A 180.000,B 0.000,C 180.000} C_DIS
LIN {X 19.469,Y 29.994,Z 57.000,A 180.000,B 0.000,C 180.000} C_DIS
LIN {X 19.469,Y 29.994,Z 52.000,A 180.000,B 0.000,C 180.000} C_DIS
LIN {X 2.500,Y 29.994,Z 52.000,A 180.000,B 0.000,C 180.000} C_DIS
LIN {X 2.500,Y 29.994,Z 45.000,A 180.000,B 0.000,C 180.000} C_DIS
LIN {X -0.010,Y 29.994,Z 45.000,A 180.000,B 0.000,C 180.000} C_DIS
; Link Move Starts
LIN {X -0.120,Y 29.994,Z 45.026,A 180.000,B 0.000,C 180.000} C_DIS
LIN {X -0.230,Y 29.994,Z 45.051,A 180.000,B 0.000,C 180.000} C_DIS
LIN {X -0.771,Y 30.307,Z 45.051,A 180.000,B 0.000,C 180.000} C_DIS
LIN {X -0.771,Y 30.932,Z 45.051,A 180.000,B 0.000,C 180.000} C_DIS
LIN {X -0.230,Y 31.244,Z 45.051,A 180.000,B 0.000,C 180.000} C_DIS
LIN {X -0.120,Y 31.244,Z 45.026,A 180.000,B 0.000,C 180.000} C_DIS
LIN {X -0.010,Y 31.244,Z 45.000,A 180.000,B 0.000,C 180.000} C_DIS
; Cutting Move Starts
LIN {X 2.500,Y 31.244,Z 45.000,A 180.000,B 0.000,C 180.000} C_DIS
LIN {X 2.500,Y 31.244,Z 52.000,A 180.000,B 0.000,C 180.000} C_DIS
LIN {X 18.468,Y 31.244,Z 52.000,A 180.000,B 0.000,C 180.000} C_DIS
LIN {X 18.468,Y 31.244,Z 57.000,A 180.000,B 0.000,C 180.000} C_DIS
LIN {X 31.156,Y 31.244,Z 57.000,A 180.000,B 0.000,C 180.000} C_DIS
LIN {X 31.156,Y 31.244,Z 52.000,A 180.000,B 0.000,C 180.000} C_DIS
LIN {X 41.844,Y 31.244,Z 52.000,A 180.000,B 0.000,C 180.000} C_DIS
LIN {X 41.844,Y 31.244,Z 57.000,A 180.000,B 0.000,C 180.000} C_DIS
LIN {X 55.220,Y 31.244,Z 57.000,A 180.000,B 0.000,C 180.000} C_DIS
LIN {X 55.220,Y 31.244,Z 62.000,A 180.000,B 0.000,C 180.000} C_DIS
LIN {X 99.780,Y 31.244,Z 62.000,A 180.000,B 0.000,C 180.000} C_DIS
LIN {X 99.780,Y 31.244,Z 57.000,A 180.000,B 0.000,C 180.000} C_DIS
LIN {X 113.156,Y 31.244,Z 57.000,A 180.000,B 0.000,C 180.000} C_DIS
LIN {X 113.156,Y 31.244,Z 52.000,A 180.000,B 0.000,C 180.000} C_DIS
LIN {X 123.844,Y 31.244,Z 52.000,A 180.000,B 0.000,C 180.000} C_DIS
LIN {X 123.844,Y 31.244,Z 57.000,A 180.000,B 0.000,C 180.000} C_DIS
LIN {X 136.532,Y 31.244,Z 57.000,A 180.000,B 0.000,C 180.000} C_DIS
LIN {X 136.532,Y 31.244,Z 52.000,A 180.000,B 0.000,C 180.000} C_DIS
LIN {X 152.500,Y 31.244,Z 52.000,A 180.000,B 0.000,C 180.000} C_DIS
LIN {X 152.500,Y 31.244,Z 45.000,A 180.000,B 0.000,C 180.000} C_DIS
LIN {X 155.010,Y 31.244,Z 45.000,A 180.000,B 0.000,C 180.000} C_DIS
; Link Move Starts
LIN {X 155.120,Y 31.244,Z 45.026,A 180.000,B 0.000,C 180.000} C_DIS
LIN {X 155.230,Y 31.244,Z 45.051,A 180.000,B 0.000,C 180.000} C_DIS
LIN {X 155.771,Y 31.557,Z 45.051,A 180.000,B 0.000,C 180.000} C_DIS
LIN {X 155.771,Y 32.182,Z 45.051,A 180.000,B 0.000,C 180.000} C_DIS
LIN {X 155.230,Y 32.494,Z 45.051,A 180.000,B 0.000,C 180.000} C_DIS
LIN {X 155.120,Y 32.494,Z 45.026,A 180.000,B 0.000,C 180.000} C_DIS
LIN {X 155.010,Y 32.494,Z 45.000,A 180.000,B 0.000,C 180.000} C_DIS
; Cutting Move Starts
LIN {X 152.500,Y 32.494,Z 45.000,A 180.000,B 0.000,C 180.000} C_DIS
LIN {X 152.500,Y 32.494,Z 52.000,A 180.000,B 0.000,C 180.000} C_DIS
LIN {X 137.489,Y 32.494,Z 52.000,A 180.000,B 0.000,C 180.000} C_DIS
LIN {X 137.486,Y 32.494,Z 57.000,A 180.000,B 0.000,C 180.000} C_DIS
LIN {X 124.839,Y 32.494,Z 57.000,A 180.000,B 0.000,C 180.000} C_DIS
LIN {X 124.839,Y 32.494,Z 52.000,A 180.000,B 0.000,C 180.000} C_DIS
LIN {X 112.161,Y 32.494,Z 52.000,A 180.000,B 0.000,C 180.000} C_DIS
LIN {X 112.161,Y 32.494,Z 57.000,A 180.000,B 0.000,C 180.000} C_DIS
LIN {X 101.030,Y 32.494,Z 57.000,A 180.000,B 0.000,C 180.000} C_DIS
LIN {X 101.030,Y 32.494,Z 62.000,A 180.000,B 0.000,C 180.000} C_DIS
LIN {X 53.970,Y 32.494,Z 62.000,A 180.000,B 0.000,C 180.000} C_DIS
LIN {X 53.968,Y 32.494,Z 57.000,A 180.000,B 0.000,C 180.000} C_DIS
LIN {X 42.839,Y 32.494,Z 57.000,A 180.000,B 0.000,C 180.000} C_DIS
LIN {X 42.839,Y 32.494,Z 52.000,A 180.000,B 0.000,C 180.000} C_DIS
LIN {X 30.161,Y 32.494,Z 52.000,A 180.000,B 0.000,C 180.000} C_DIS
LIN {X 30.161,Y 32.494,Z 57.000,A 180.000,B 0.000,C 180.000} C_DIS
LIN {X 17.511,Y 32.494,Z 57.000,A 180.000,B 0.000,C 180.000} C_DIS
LIN {X 17.511,Y 32.494,Z 52.000,A 180.000,B 0.000,C 180.000} C_DIS
LIN {X 2.500,Y 32.494,Z 52.000,A 180.000,B 0.000,C 180.000} C_DIS
LIN {X 2.500,Y 32.494,Z 45.000,A 180.000,B 0.000,C 180.000} C_DIS
LIN {X -0.010,Y 32.494,Z 45.000,A 180.000,B 0.000,C 180.000} C_DIS
; Link Move Starts
LIN {X -0.120,Y 32.494,Z 45.026,A 180.000,B 0.000,C 180.000} C_DIS
LIN {X -0.230,Y 32.494,Z 45.051,A 180.000,B 0.000,C 180.000} C_DIS
LIN {X -0.771,Y 32.807,Z 45.051,A 180.000,B 0.000,C 180.000} C_DIS
LIN {X -0.771,Y 33.432,Z 45.051,A 180.000,B 0.000,C 180.000} C_DIS
LIN {X -0.230,Y 33.744,Z 45.051,A 180.000,B 0.000,C 180.000} C_DIS
LIN {X -0.120,Y 33.744,Z 45.026,A 180.000,B 0.000,C 180.000} C_DIS
LIN {X -0.010,Y 33.744,Z 45.000,A 180.000,B 0.000,C 180.000} C_DIS
; Cutting Move Starts
LIN {X 2.500,Y 33.744,Z 45.000,A 180.000,B 0.000,C 180.000} C_DIS
LIN {X 2.500,Y 33.744,Z 52.000,A 180.000,B 0.000,C 180.000} C_DIS
LIN {X 16.593,Y 33.744,Z 52.000,A 180.000,B 0.000,C 180.000} C_DIS
LIN {X 16.593,Y 33.744,Z 57.000,A 180.000,B 0.000,C 180.000} C_DIS
LIN {X 29.526,Y 33.744,Z 57.000,A 180.000,B 0.000,C 180.000} C_DIS
LIN {X 29.526,Y 33.744,Z 52.000,A 180.000,B 0.000,C 180.000} C_DIS
LIN {X 43.474,Y 33.744,Z 52.000,A 180.000,B 0.000,C 180.000} C_DIS
LIN {X 43.474,Y 33.744,Z 57.000,A 180.000,B 0.000,C 180.000} C_DIS
LIN {X 52.720,Y 33.744,Z 57.000,A 180.000,B 0.000,C 180.000} C_DIS
LIN {X 52.720,Y 33.744,Z 62.000,A 180.000,B 0.000,C 180.000} C_DIS
LIN {X 102.280,Y 33.744,Z 62.000,A 180.000,B 0.000,C 180.000} C_DIS
LIN {X 102.280,Y 33.744,Z 57.000,A 180.000,B 0.000,C 180.000} C_DIS
LIN {X 111.526,Y 33.744,Z 57.000,A 180.000,B 0.000,C 180.000} C_DIS
LIN {X 111.526,Y 33.744,Z 52.000,A 180.000,B 0.000,C 180.000} C_DIS
LIN {X 125.474,Y 33.744,Z 52.000,A 180.000,B 0.000,C 180.000} C_DIS
LIN {X 125.474,Y 33.744,Z 57.000,A 180.000,B 0.000,C 180.000} C_DIS
LIN {X 138.404,Y 33.744,Z 57.000,A 180.000,B 0.000,C 180.000} C_DIS
LIN {X 138.407,Y 33.744,Z 52.000,A 180.000,B 0.000,C 180.000} C_DIS
LIN {X 152.500,Y 33.744,Z 52.000,A 180.000,B 0.000,C 180.000} C_DIS
LIN {X 152.500,Y 33.744,Z 45.000,A 180.000,B 0.000,C 180.000} C_DIS
LIN {X 155.010,Y 33.744,Z 45.000,A 180.000,B 0.000,C 180.000} C_DIS
; Link Move Starts
LIN {X 155.120,Y 33.744,Z 45.026,A 180.000,B 0.000,C 180.000} C_DIS
LIN {X 155.230,Y 33.744,Z 45.051,A 180.000,B 0.000,C 180.000} C_DIS
LIN {X 155.771,Y 34.056,Z 45.051,A 180.000,B 0.000,C 180.000} C_DIS
LIN {X 155.771,Y 34.681,Z 45.051,A 180.000,B 0.000,C 180.000} C_DIS
LIN {X 155.230,Y 34.994,Z 45.051,A 180.000,B 0.000,C 180.000} C_DIS
LIN {X 155.120,Y 34.994,Z 45.026,A 180.000,B 0.000,C 180.000} C_DIS
LIN {X 155.010,Y 34.994,Z 45.000,A 180.000,B 0.000,C 180.000} C_DIS
; Cutting Move Starts
LIN {X 152.500,Y 34.994,Z 45.000,A 180.000,B 0.000,C 180.000} C_DIS
LIN {X 152.500,Y 34.994,Z 52.000,A 180.000,B 0.000,C 180.000} C_DIS
LIN {X 139.287,Y 34.994,Z 52.000,A 180.000,B 0.000,C 180.000} C_DIS
LIN {X 139.287,Y 34.994,Z 57.000,A 180.000,B 0.000,C 180.000} C_DIS
LIN {X 125.843,Y 34.994,Z 57.000,A 180.000,B 0.000,C 180.000} C_DIS
LIN {X 125.843,Y 34.994,Z 52.000,A 180.000,B 0.000,C 180.000} C_DIS
LIN {X 111.157,Y 34.994,Z 52.000,A 180.000,B 0.000,C 180.000} C_DIS
LIN {X 111.157,Y 34.994,Z 57.000,A 180.000,B 0.000,C 180.000} C_DIS
LIN {X 103.529,Y 34.994,Z 57.000,A 180.000,B 0.000,C 180.000} C_DIS
LIN {X 103.529,Y 34.994,Z 62.000,A 180.000,B 0.000,C 180.000} C_DIS
LIN {X 51.471,Y 34.994,Z 62.000,A 180.000,B 0.000,C 180.000} C_DIS
LIN {X 51.471,Y 34.994,Z 57.000,A 180.000,B 0.000,C 180.000} C_DIS
LIN {X 43.843,Y 34.994,Z 57.000,A 180.000,B 0.000,C 180.000} C_DIS
LIN {X 43.843,Y 34.994,Z 52.000,A 180.000,B 0.000,C 180.000} C_DIS
LIN {X 29.157,Y 34.994,Z 52.000,A 180.000,B 0.000,C 180.000} C_DIS
LIN {X 29.157,Y 34.994,Z 57.000,A 180.000,B 0.000,C 180.000} C_DIS
LIN {X 15.713,Y 34.994,Z 57.000,A 180.000,B 0.000,C 180.000} C_DIS
LIN {X 15.713,Y 34.994,Z 52.000,A 180.000,B 0.000,C 180.000} C_DIS
LIN {X 2.500,Y 34.994,Z 52.000,A 180.000,B 0.000,C 180.000} C_DIS
LIN {X 2.500,Y 34.994,Z 45.000,A 180.000,B 0.000,C 180.000} C_DIS
LIN {X -0.010,Y 34.994,Z 45.000,A 180.000,B 0.000,C 180.000} C_DIS
; Link Move Starts
LIN {X -0.120,Y 34.994,Z 45.026,A 180.000,B 0.000,C 180.000} C_DIS
LIN {X -0.230,Y 34.994,Z 45.051,A 180.000,B 0.000,C 180.000} C_DIS
LIN {X -0.771,Y 35.306,Z 45.051,A 180.000,B 0.000,C 180.000} C_DIS
LIN {X -0.771,Y 35.931,Z 45.051,A 180.000,B 0.000,C 180.000} C_DIS
LIN {X -0.230,Y 36.244,Z 45.051,A 180.000,B 0.000,C 180.000} C_DIS
LIN {X -0.120,Y 36.244,Z 45.026,A 180.000,B 0.000,C 180.000} C_DIS
LIN {X -0.010,Y 36.244,Z 45.000,A 180.000,B 0.000,C 180.000} C_DIS
; Cutting Move Starts
LIN {X 2.500,Y 36.244,Z 45.000,A 180.000,B 0.000,C 180.000} C_DIS
LIN {X 2.500,Y 36.244,Z 52.000,A 180.000,B 0.000,C 180.000} C_DIS
LIN {X 14.870,Y 36.244,Z 52.000,A 180.000,B 0.000,C 180.000} C_DIS
LIN {X 14.870,Y 36.244,Z 57.000,A 180.000,B 0.000,C 180.000} C_DIS
LIN {X 29.006,Y 36.244,Z 57.000,A 180.000,B 0.000,C 180.000} C_DIS
LIN {X 29.009,Y 36.244,Z 52.000,A 180.000,B 0.000,C 180.000} C_DIS
LIN {X 43.991,Y 36.244,Z 52.000,A 180.000,B 0.000,C 180.000} C_DIS
LIN {X 43.991,Y 36.244,Z 57.000,A 180.000,B 0.000,C 180.000} C_DIS
LIN {X 50.221,Y 36.244,Z 57.000,A 180.000,B 0.000,C 180.000} C_DIS
LIN {X 50.221,Y 36.244,Z 62.000,A 180.000,B 0.000,C 180.000} C_DIS
LIN {X 86.761,Y 36.244,Z 62.000,A 180.000,B 0.000,C 180.000} C_DIS
LIN {X 86.762,Y 36.244,Z 72.976,A 180.000,B 0.000,C 180.000} C_DIS
LIN {X 86.780,Y 36.244,Z 73.031,A 180.000,B 0.000,C 180.000} C_DIS
LIN {X 86.824,Y 36.244,Z 73.076,A 180.000,B 0.000,C 180.000} C_DIS
LIN {X 86.907,Y 36.244,Z 73.113,A 180.000,B 0.000,C 180.000} C_DIS
LIN {X 87.044,Y 36.244,Z 73.138,A 180.000,B 0.000,C 180.000} C_DIS
LIN {X 87.247,Y 36.244,Z 73.142,A 180.000,B 0.000,C 180.000} C_DIS
LIN {X 87.514,Y 36.244,Z 73.120,A 180.000,B 0.000,C 180.000} C_DIS
LIN {X 87.926,Y 36.244,Z 73.055,A 180.000,B 0.000,C 180.000} C_DIS
LIN {X 88.473,Y 36.244,Z 72.936,A 180.000,B 0.000,C 180.000} C_DIS
LIN {X 89.178,Y 36.244,Z 72.751,A 180.000,B 0.000,C 180.000} C_DIS
LIN {X 90.042,Y 36.244,Z 72.492,A 180.000,B 0.000,C 180.000} C_DIS
LIN {X 91.058,Y 36.244,Z 72.155,A 180.000,B 0.000,C 180.000} C_DIS
LIN {X 91.058,Y 36.244,Z 67.085,A 180.000,B 0.000,C 180.000} C_DIS
LIN {X 91.201,Y 36.244,Z 67.108,A 180.000,B 0.000,C 180.000} C_DIS
LIN {X 91.681,Y 36.244,Z 67.186,A 180.000,B 0.000,C 180.000} C_DIS
LIN {X 92.354,Y 36.244,Z 67.226,A 180.000,B 0.000,C 180.000} C_DIS
LIN {X 92.910,Y 36.244,Z 67.213,A 180.000,B 0.000,C 180.000} C_DIS
LIN {X 93.155,Y 36.244,Z 67.200,A 180.000,B 0.000,C 180.000} C_DIS
LIN {X 93.790,Y 36.244,Z 67.116,A 180.000,B 0.000,C 180.000} C_DIS
LIN {X 94.507,Y 36.244,Z 66.951,A 180.000,B 0.000,C 180.000} C_DIS
LIN {X 95.099,Y 36.244,Z 66.758,A 180.000,B 0.000,C 180.000} C_DIS
LIN {X 95.250,Y 36.244,Z 66.699,A 180.000,B 0.000,C 180.000} C_DIS
LIN {X 95.813,Y 36.244,Z 66.416,A 180.000,B 0.000,C 180.000} C_DIS
LIN {X 96.049,Y 36.244,Z 66.292,A 180.000,B 0.000,C 180.000} C_DIS
LIN {X 96.689,Y 36.244,Z 65.813,A 180.000,B 0.000,C 180.000} C_DIS
LIN {X 96.806,Y 36.244,Z 65.702,A 180.000,B 0.000,C 180.000} C_DIS
LIN {X 97.154,Y 36.244,Z 65.321,A 180.000,B 0.000,C 180.000} C_DIS
LIN {X 97.505,Y 36.244,Z 64.817,A 180.000,B 0.000,C 180.000} C_DIS
LIN {X 97.545,Y 36.244,Z 64.742,A 180.000,B 0.000,C 180.000} C_DIS
LIN {X 97.742,Y 36.244,Z 64.310,A 180.000,B 0.000,C 180.000} C_DIS
LIN {X 97.878,Y 36.244,Z 63.788,A 180.000,B 0.000,C 180.000} C_DIS
LIN {X 97.923,Y 36.244,Z 63.286,A 180.000,B 0.000,C 180.000} C_DIS
LIN {X 97.926,Y 36.244,Z 62.000,A 180.000,B 0.000,C 180.000} C_DIS
LIN {X 104.779,Y 36.244,Z 62.000,A 180.000,B 0.000,C 180.000} C_DIS
LIN {X 104.779,Y 36.244,Z 57.000,A 180.000,B 0.000,C 180.000} C_DIS
LIN {X 111.007,Y 36.244,Z 57.000,A 180.000,B 0.000,C 180.000} C_DIS
LIN {X 111.009,Y 36.244,Z 52.000,A 180.000,B 0.000,C 180.000} C_DIS
LIN {X 125.989,Y 36.244,Z 52.000,A 180.000,B 0.000,C 180.000} C_DIS
LIN {X 125.991,Y 36.244,Z 57.000,A 180.000,B 0.000,C 180.000} C_DIS
LIN {X 140.130,Y 36.244,Z 57.000,A 180.000,B 0.000,C 180.000} C_DIS
LIN {X 140.130,Y 36.244,Z 52.000,A 180.000,B 0.000,C 180.000} C_DIS
LIN {X 152.500,Y 36.244,Z 52.000,A 180.000,B 0.000,C 180.000} C_DIS
LIN {X 152.500,Y 36.244,Z 45.000,A 180.000,B 0.000,C 180.000} C_DIS
LIN {X 155.010,Y 36.244,Z 45.000,A 180.000,B 0.000,C 180.000} C_DIS
; Link Move Starts
LIN {X 155.120,Y 36.244,Z 45.026,A 180.000,B 0.000,C 180.000} C_DIS
LIN {X 155.230,Y 36.244,Z 45.051,A 180.000,B 0.000,C 180.000} C_DIS
LIN {X 155.771,Y 36.556,Z 45.051,A 180.000,B 0.000,C 180.000} C_DIS
LIN {X 155.771,Y 37.181,Z 45.051,A 180.000,B 0.000,C 180.000} C_DIS
LIN {X 155.230,Y 37.494,Z 45.051,A 180.000,B 0.000,C 180.000} C_DIS
LIN {X 155.120,Y 37.494,Z 45.026,A 180.000,B 0.000,C 180.000} C_DIS
LIN {X 155.010,Y 37.494,Z 45.000,A 180.000,B 0.000,C 180.000} C_DIS
; Cutting Move Starts
LIN {X 152.500,Y 37.494,Z 45.000,A 180.000,B 0.000,C 180.000} C_DIS
LIN {X 152.500,Y 37.494,Z 52.000,A 180.000,B 0.000,C 180.000} C_DIS
LIN {X 140.939,Y 37.494,Z 52.000,A 180.000,B 0.000,C 180.000} C_DIS
LIN {X 140.939,Y 37.494,Z 57.000,A 180.000,B 0.000,C 180.000} C_DIS
LIN {X 125.931,Y 37.494,Z 57.000,A 180.000,B 0.000,C 180.000} C_DIS
LIN {X 125.931,Y 37.494,Z 52.000,A 180.000,B 0.000,C 180.000} C_DIS
LIN {X 111.069,Y 37.494,Z 52.000,A 180.000,B 0.000,C 180.000} C_DIS
LIN {X 111.065,Y 37.494,Z 57.000,A 180.000,B 0.000,C 180.000} C_DIS
LIN {X 106.029,Y 37.494,Z 57.000,A 180.000,B 0.000,C 180.000} C_DIS
LIN {X 106.029,Y 37.494,Z 62.000,A 180.000,B 0.000,C 180.000} C_DIS
LIN {X 99.984,Y 37.494,Z 62.000,A 180.000,B 0.000,C 180.000} C_DIS
LIN {X 99.982,Y 37.494,Z 63.277,A 180.000,B 0.000,C 180.000} C_DIS
LIN {X 99.948,Y 37.494,Z 63.790,A 180.000,B 0.000,C 180.000} C_DIS
LIN {X 99.849,Y 37.494,Z 64.306,A 180.000,B 0.000,C 180.000} C_DIS
LIN {X 99.686,Y 37.494,Z 64.820,A 180.000,B 0.000,C 180.000} C_DIS
LIN {X 99.456,Y 37.494,Z 65.312,A 180.000,B 0.000,C 180.000} C_DIS
LIN {X 99.135,Y 37.494,Z 65.816,A 180.000,B 0.000,C 180.000} C_DIS
LIN {X 98.752,Y 37.494,Z 66.298,A 180.000,B 0.000,C 180.000} C_DIS
LIN {X 98.473,Y 37.494,Z 66.568,A 180.000,B 0.000,C 180.000} C_DIS
LIN {X 98.267,Y 37.494,Z 66.760,A 180.000,B 0.000,C 180.000} C_DIS
LIN {X 97.825,Y 37.494,Z 67.108,A 180.000,B 0.000,C 180.000} C_DIS
LIN {X 97.686,Y 37.494,Z 67.204,A 180.000,B 0.000,C 180.000} C_DIS
LIN {X 97.047,Y 37.494,Z 67.586,A 180.000,B 0.000,C 180.000} C_DIS
LIN {X 96.901,Y 37.494,Z 67.656,A 180.000,B 0.000,C 180.000} C_DIS
LIN {X 96.301,Y 37.494,Z 67.923,A 180.000,B 0.000,C 180.000} C_DIS
LIN {X 96.033,Y 37.494,Z 68.024,A 180.000,B 0.000,C 180.000} C_DIS
LIN {X 95.583,Y 37.494,Z 68.168,A 180.000,B 0.000,C 180.000} C_DIS
LIN {X 94.919,Y 37.494,Z 68.345,A 180.000,B 0.000,C 180.000} C_DIS
LIN {X 94.649,Y 37.494,Z 68.398,A 180.000,B 0.000,C 180.000} C_DIS
LIN {X 94.234,Y 37.494,Z 68.469,A 180.000,B 0.000,C 180.000} C_DIS
LIN {X 93.618,Y 37.494,Z 68.544,A 180.000,B 0.000,C 180.000} C_DIS
LIN {X 92.999,Y 37.494,Z 68.587,A 180.000,B 0.000,C 180.000} C_DIS
LIN {X 92.372,Y 37.494,Z 68.597,A 180.000,B 0.000,C 180.000} C_DIS
LIN {X 91.763,Y 37.494,Z 68.574,A 180.000,B 0.000,C 180.000} C_DIS
LIN {X 91.761,Y 37.494,Z 72.156,A 180.000,B 0.000,C 180.000} C_DIS
LIN {X 90.221,Y 37.494,Z 72.793,A 180.000,B 0.000,C 180.000} C_DIS
LIN {X 88.950,Y 37.494,Z 73.292,A 180.000,B 0.000,C 180.000} C_DIS
LIN {X 87.763,Y 37.494,Z 73.729,A 180.000,B 0.000,C 180.000} C_DIS
LIN {X 86.695,Y 37.494,Z 74.094,A 180.000,B 0.000,C 180.000} C_DIS
LIN {X 85.830,Y 37.494,Z 74.364,A 180.000,B 0.000,C 180.000} C_DIS
LIN {X 83.242,Y 37.494,Z 74.362,A 180.000,B 0.000,C 180.000} C_DIS
LIN {X 83.129,Y 37.494,Z 74.083,A 180.000,B 0.000,C 180.000} C_DIS
LIN {X 83.071,Y 37.494,Z 73.871,A 180.000,B 0.000,C 180.000} C_DIS
LIN {X 83.056,Y 37.494,Z 73.727,A 180.000,B 0.000,C 180.000} C_DIS
LIN {X 83.056,Y 37.494,Z 62.000,A 180.000,B 0.000,C 180.000} C_DIS
LIN {X 48.971,Y 37.494,Z 62.000,A 180.000,B 0.000,C 180.000} C_DIS
LIN {X 48.971,Y 37.494,Z 57.000,A 180.000,B 0.000,C 180.000} C_DIS
LIN {X 43.931,Y 37.494,Z 57.000,A 180.000,B 0.000,C 180.000} C_DIS
LIN {X 43.931,Y 37.494,Z 52.000,A 180.000,B 0.000,C 180.000} C_DIS
LIN {X 29.069,Y 37.494,Z 52.000,A 180.000,B 0.000,C 180.000} C_DIS
LIN {X 29.068,Y 37.494,Z 57.000,A 180.000,B 0.000,C 180.000} C_DIS
LIN {X 14.061,Y 37.494,Z 57.000,A 180.000,B 0.000,C 180.000} C_DIS
LIN {X 14.061,Y 37.494,Z 52.000,A 180.000,B 0.000,C 180.000} C_DIS
LIN {X 2.500,Y 37.494,Z 52.000,A 180.000,B 0.000,C 180.000} C_DIS
LIN {X 2.500,Y 37.494,Z 45.000,A 180.000,B 0.000,C 180.000} C_DIS
LIN {X -0.010,Y 37.494,Z 45.000,A 180.000,B 0.000,C 180.000} C_DIS
; Link Move Starts
LIN {X -0.120,Y 37.494,Z 45.026,A 180.000,B 0.000,C 180.000} C_DIS
LIN {X -0.230,Y 37.494,Z 45.051,A 180.000,B 0.000,C 180.000} C_DIS
LIN {X -0.771,Y 37.806,Z 45.051,A 180.000,B 0.000,C 180.000} C_DIS
LIN {X -0.771,Y 38.431,Z 45.051,A 180.000,B 0.000,C 180.000} C_DIS
LIN {X -0.230,Y 38.744,Z 45.051,A 180.000,B 0.000,C 180.000} C_DIS
LIN {X -0.120,Y 38.744,Z 45.026,A 180.000,B 0.000,C 180.000} C_DIS
LIN {X -0.010,Y 38.744,Z 45.000,A 180.000,B 0.000,C 180.000} C_DIS
; Cutting Move Starts
LIN {X 2.500,Y 38.744,Z 45.000,A 180.000,B 0.000,C 180.000} C_DIS
LIN {X 2.500,Y 38.744,Z 52.000,A 180.000,B 0.000,C 180.000} C_DIS
LIN {X 13.292,Y 38.744,Z 52.000,A 180.000,B 0.000,C 180.000} C_DIS
LIN {X 13.293,Y 38.744,Z 57.000,A 180.000,B 0.000,C 180.000} C_DIS
LIN {X 29.347,Y 38.744,Z 57.000,A 180.000,B 0.000,C 180.000} C_DIS
LIN {X 29.347,Y 38.744,Z 52.000,A 180.000,B 0.000,C 180.000} C_DIS
LIN {X 43.653,Y 38.744,Z 52.000,A 180.000,B 0.000,C 180.000} C_DIS
LIN {X 43.653,Y 38.744,Z 57.000,A 180.000,B 0.000,C 180.000} C_DIS
LIN {X 47.721,Y 38.744,Z 57.000,A 180.000,B 0.000,C 180.000} C_DIS
LIN {X 47.721,Y 38.744,Z 62.000,A 180.000,B 0.000,C 180.000} C_DIS
LIN {X 79.351,Y 38.744,Z 62.000,A 180.000,B 0.000,C 180.000} C_DIS
LIN {X 79.353,Y 38.744,Z 71.137,A 180.000,B 0.000,C 180.000} C_DIS
LIN {X 79.374,Y 38.744,Z 71.218,A 180.000,B 0.000,C 180.000} C_DIS
LIN {X 79.443,Y 38.744,Z 71.347,A 180.000,B 0.000,C 180.000} C_DIS
LIN {X 79.574,Y 38.744,Z 71.528,A 180.000,B 0.000,C 180.000} C_DIS
LIN {X 79.836,Y 38.744,Z 71.833,A 180.000,B 0.000,C 180.000} C_DIS
LIN {X 81.216,Y 38.744,Z 73.292,A 180.000,B 0.000,C 180.000} C_DIS
LIN {X 82.198,Y 38.744,Z 74.361,A 180.000,B 0.000,C 180.000} C_DIS
LIN {X 86.871,Y 38.744,Z 74.364,A 180.000,B 0.000,C 180.000} C_DIS
LIN {X 92.184,Y 38.744,Z 72.155,A 180.000,B 0.000,C 180.000} C_DIS
LIN {X 92.185,Y 38.744,Z 69.433,A 180.000,B 0.000,C 180.000} C_DIS
LIN {X 92.314,Y 38.744,Z 69.436,A 180.000,B 0.000,C 180.000} C_DIS
LIN {X 92.868,Y 38.744,Z 69.433,A 180.000,B 0.000,C 180.000} C_DIS
LIN {X 93.418,Y 38.744,Z 69.412,A 180.000,B 0.000,C 180.000} C_DIS
LIN {X 93.988,Y 38.744,Z 69.371,A 180.000,B 0.000,C 180.000} C_DIS
LIN {X 94.575,Y 38.744,Z 69.309,A 180.000,B 0.000,C 180.000} C_DIS
LIN {X 95.141,Y 38.744,Z 69.216,A 180.000,B 0.000,C 180.000} C_DIS
LIN {X 95.592,Y 38.744,Z 69.127,A 180.000,B 0.000,C 180.000} C_DIS
LIN {X 95.976,Y 38.744,Z 69.043,A 180.000,B 0.000,C 180.000} C_DIS
LIN {X 96.432,Y 38.744,Z 68.915,A 180.000,B 0.000,C 180.000} C_DIS
LIN {X 96.978,Y 38.744,Z 68.739,A 180.000,B 0.000,C 180.000} C_DIS
LIN {X 97.145,Y 38.744,Z 68.678,A 180.000,B 0.000,C 180.000} C_DIS
LIN {X 97.868,Y 38.744,Z 68.368,A 180.000,B 0.000,C 180.000} C_DIS
LIN {X 98.494,Y 38.744,Z 68.025,A 180.000,B 0.000,C 180.000} C_DIS
LIN {X 98.650,Y 38.744,Z 67.927,A 180.000,B 0.000,C 180.000} C_DIS
LIN {X 99.083,Y 38.744,Z 67.627,A 180.000,B 0.000,C 180.000} C_DIS
LIN {X 99.602,Y 38.744,Z 67.202,A 180.000,B 0.000,C 180.000} C_DIS
LIN {X 100.028,Y 38.744,Z 66.763,A 180.000,B 0.000,C 180.000} C_DIS
LIN {X 100.410,Y 38.744,Z 66.293,A 180.000,B 0.000,C 180.000} C_DIS
LIN {X 100.714,Y 38.744,Z 65.822,A 180.000,B 0.000,C 180.000} C_DIS
LIN {X 100.964,Y 38.744,Z 65.326,A 180.000,B 0.000,C 180.000} C_DIS
LIN {X 101.160,Y 38.744,Z 64.821,A 180.000,B 0.000,C 180.000} C_DIS
LIN {X 101.298,Y 38.744,Z 64.317,A 180.000,B 0.000,C 180.000} C_DIS
LIN {X 101.384,Y 38.744,Z 63.801,A 180.000,B 0.000,C 180.000} C_DIS
LIN {X 101.415,Y 38.744,Z 63.292,A 180.000,B 0.000,C 180.000} C_DIS
LIN {X 101.417,Y 38.744,Z 62.000,A 180.000,B 0.000,C 180.000} C_DIS
LIN {X 107.276,Y 38.744,Z 62.000,A 180.000,B 0.000,C 180.000} C_DIS
LIN {X 107.279,Y 38.744,Z 57.000,A 180.000,B 0.000,C 180.000} C_DIS
LIN {X 111.343,Y 38.744,Z 57.000,A 180.000,B 0.000,C 180.000} C_DIS
LIN {X 111.347,Y 38.744,Z 52.000,A 180.000,B 0.000,C 180.000} C_DIS
LIN {X 125.652,Y 38.744,Z 52.000,A 180.000,B 0.000,C 180.000} C_DIS
LIN {X 125.653,Y 38.744,Z 57.000,A 180.000,B 0.000,C 180.000} C_DIS
LIN {X 141.707,Y 38.744,Z 57.000,A 180.000,B 0.000,C 180.000} C_DIS
LIN {X 141.707,Y 38.744,Z 52.000,A 180.000,B 0.000,C 180.000} C_DIS
LIN {X 152.500,Y 38.744,Z 52.000,A 180.000,B 0.000,C 180.000} C_DIS
LIN {X 152.500,Y 38.744,Z 45.000,A 180.000,B 0.000,C 180.000} C_DIS
LIN {X 155.010,Y 38.744,Z 45.000,A 180.000,B 0.000,C 180.000} C_DIS
; Link Move Starts
LIN {X 155.120,Y 38.744,Z 45.026,A 180.000,B 0.000,C 180.000} C_DIS
LIN {X 155.230,Y 38.744,Z 45.051,A 180.000,B 0.000,C 180.000} C_DIS
LIN {X 155.771,Y 39.056,Z 45.051,A 180.000,B 0.000,C 180.000} C_DIS
LIN {X 155.771,Y 39.681,Z 45.051,A 180.000,B 0.000,C 180.000} C_DIS
LIN {X 155.230,Y 39.993,Z 45.051,A 180.000,B 0.000,C 180.000} C_DIS
LIN {X 155.120,Y 39.993,Z 45.026,A 180.000,B 0.000,C 180.000} C_DIS
LIN {X 155.010,Y 39.993,Z 45.000,A 180.000,B 0.000,C 180.000} C_DIS
; Cutting Move Starts
LIN {X 152.500,Y 39.993,Z 45.000,A 180.000,B 0.000,C 180.000} C_DIS
LIN {X 152.500,Y 39.993,Z 52.000,A 180.000,B 0.000,C 180.000} C_DIS
LIN {X 142.443,Y 39.993,Z 52.000,A 180.000,B 0.000,C 180.000} C_DIS
LIN {X 142.443,Y 39.993,Z 57.000,A 180.000,B 0.000,C 180.000} C_DIS
LIN {X 125.132,Y 39.993,Z 57.000,A 180.000,B 0.000,C 180.000} C_DIS
LIN {X 125.132,Y 39.993,Z 52.000,A 180.000,B 0.000,C 180.000} C_DIS
LIN {X 111.868,Y 39.993,Z 52.000,A 180.000,B 0.000,C 180.000} C_DIS
LIN {X 111.868,Y 39.993,Z 57.000,A 180.000,B 0.000,C 180.000} C_DIS
LIN {X 108.529,Y 39.993,Z 57.000,A 180.000,B 0.000,C 180.000} C_DIS
LIN {X 108.529,Y 39.993,Z 62.000,A 180.000,B 0.000,C 180.000} C_DIS
LIN {X 102.494,Y 39.993,Z 62.000,A 180.000,B 0.000,C 180.000} C_DIS
LIN {X 102.490,Y 39.993,Z 63.332,A 180.000,B 0.000,C 180.000} C_DIS
LIN {X 102.463,Y 39.993,Z 63.818,A 180.000,B 0.000,C 180.000} C_DIS
LIN {X 102.390,Y 39.993,Z 64.310,A 180.000,B 0.000,C 180.000} C_DIS
LIN {X 102.262,Y 39.993,Z 64.830,A 180.000,B 0.000,C 180.000} C_DIS
LIN {X 102.088,Y 39.993,Z 65.332,A 180.000,B 0.000,C 180.000} C_DIS
LIN {X 101.865,Y 39.993,Z 65.825,A 180.000,B 0.000,C 180.000} C_DIS
LIN {X 101.596,Y 39.993,Z 66.304,A 180.000,B 0.000,C 180.000} C_DIS
LIN {X 101.278,Y 39.993,Z 66.765,A 180.000,B 0.000,C 180.000} C_DIS
LIN {X 100.904,Y 39.993,Z 67.205,A 180.000,B 0.000,C 180.000} C_DIS
LIN {X 100.480,Y 39.993,Z 67.629,A 180.000,B 0.000,C 180.000} C_DIS
LIN {X 100.072,Y 39.993,Z 67.969,A 180.000,B 0.000,C 180.000} C_DIS
LIN {X 99.979,Y 39.993,Z 68.039,A 180.000,B 0.000,C 180.000} C_DIS
LIN {X 99.469,Y 39.993,Z 68.393,A 180.000,B 0.000,C 180.000} C_DIS
LIN {X 98.892,Y 39.993,Z 68.721,A 180.000,B 0.000,C 180.000} C_DIS
LIN {X 98.437,Y 39.993,Z 68.935,A 180.000,B 0.000,C 180.000} C_DIS
LIN {X 98.188,Y 39.993,Z 69.044,A 180.000,B 0.000,C 180.000} C_DIS
LIN {X 97.698,Y 39.993,Z 69.226,A 180.000,B 0.000,C 180.000} C_DIS
LIN {X 97.415,Y 39.993,Z 69.322,A 180.000,B 0.000,C 180.000} C_DIS
LIN {X 96.925,Y 39.993,Z 69.459,A 180.000,B 0.000,C 180.000} C_DIS
LIN {X 96.522,Y 39.993,Z 69.563,A 180.000,B 0.000,C 180.000} C_DIS
LIN {X 95.827,Y 39.993,Z 69.695,A 180.000,B 0.000,C 180.000} C_DIS
LIN {X 95.365,Y 39.993,Z 69.771,A 180.000,B 0.000,C 180.000} C_DIS
LIN {X 94.720,Y 39.993,Z 69.842,A 180.000,B 0.000,C 180.000} C_DIS
LIN {X 94.150,Y 39.993,Z 69.892,A 180.000,B 0.000,C 180.000} C_DIS
LIN {X 93.595,Y 39.993,Z 69.927,A 180.000,B 0.000,C 180.000} C_DIS
LIN {X 93.105,Y 39.993,Z 69.944,A 180.000,B 0.000,C 180.000} C_DIS
LIN {X 92.606,Y 39.993,Z 69.950,A 180.000,B 0.000,C 180.000} C_DIS
LIN {X 92.606,Y 39.993,Z 72.155,A 180.000,B 0.000,C 180.000} C_DIS
LIN {X 87.296,Y 39.993,Z 74.364,A 180.000,B 0.000,C 180.000} C_DIS
LIN {X 82.062,Y 39.993,Z 74.362,A 180.000,B 0.000,C 180.000} C_DIS
LIN {X 81.236,Y 39.993,Z 73.618,A 180.000,B 0.000,C 180.000} C_DIS
LIN {X 80.506,Y 39.993,Z 72.993,A 180.000,B 0.000,C 180.000} C_DIS
LIN {X 79.818,Y 39.993,Z 72.438,A 180.000,B 0.000,C 180.000} C_DIS
LIN {X 79.166,Y 39.993,Z 71.946,A 180.000,B 0.000,C 180.000} C_DIS
LIN {X 78.549,Y 39.993,Z 71.516,A 180.000,B 0.000,C 180.000} C_DIS
LIN {X 78.001,Y 39.993,Z 71.166,A 180.000,B 0.000,C 180.000} C_DIS
LIN {X 77.520,Y 39.993,Z 70.886,A 180.000,B 0.000,C 180.000} C_DIS
LIN {X 77.041,Y 39.993,Z 70.634,A 180.000,B 0.000,C 180.000} C_DIS
LIN {X 76.622,Y 39.993,Z 70.439,A 180.000,B 0.000,C 180.000} C_DIS
LIN {X 76.219,Y 39.993,Z 70.276,A 180.000,B 0.000,C 180.000} C_DIS
LIN {X 75.835,Y 39.993,Z 70.146,A 180.000,B 0.000,C 180.000} C_DIS
LIN {X 75.648,Y 39.993,Z 70.083,A 180.000,B 0.000,C 180.000} C_DIS
LIN {X 75.646,Y 39.993,Z 62.000,A 180.000,B 0.000,C 180.000} C_DIS
LIN {X 46.471,Y 39.993,Z 62.000,A 180.000,B 0.000,C 180.000} C_DIS
LIN {X 46.471,Y 39.993,Z 57.000,A 180.000,B 0.000,C 180.000} C_DIS
LIN {X 43.132,Y 39.993,Z 57.000,A 180.000,B 0.000,C 180.000} C_DIS
LIN {X 43.132,Y 39.993,Z 52.000,A 180.000,B 0.000,C 180.000} C_DIS
LIN {X 29.868,Y 39.993,Z 52.000,A 180.000,B 0.000,C 180.000} C_DIS
LIN {X 29.868,Y 39.993,Z 57.000,A 180.000,B 0.000,C 180.000} C_DIS
LIN {X 12.557,Y 39.993,Z 57.000,A 180.000,B 0.000,C 180.000} C_DIS
LIN {X 12.557,Y 39.993,Z 52.000,A 180.000,B 0.000,C 180.000} C_DIS
LIN {X 2.500,Y 39.993,Z 52.000,A 180.000,B 0.000,C 180.000} C_DIS
LIN {X 2.500,Y 39.993,Z 45.000,A 180.000,B 0.000,C 180.000} C_DIS
LIN {X -0.010,Y 39.993,Z 45.000,A 180.000,B 0.000,C 180.000} C_DIS
; Link Move Starts
LIN {X -0.120,Y 39.993,Z 45.026,A 180.000,B 0.000,C 180.000} C_DIS
LIN {X -0.230,Y 39.993,Z 45.051,A 180.000,B 0.000,C 180.000} C_DIS
LIN {X -0.771,Y 40.306,Z 45.051,A 180.000,B 0.000,C 180.000} C_DIS
LIN {X -0.771,Y 40.931,Z 45.051,A 180.000,B 0.000,C 180.000} C_DIS
LIN {X -0.230,Y 41.243,Z 45.051,A 180.000,B 0.000,C 180.000} C_DIS
LIN {X -0.120,Y 41.243,Z 45.026,A 180.000,B 0.000,C 180.000} C_DIS
LIN {X -0.010,Y 41.243,Z 45.000,A 180.000,B 0.000,C 180.000} C_DIS
; Cutting Move Starts
LIN {X 2.500,Y 41.243,Z 45.000,A 180.000,B 0.000,C 180.000} C_DIS
LIN {X 2.500,Y 41.243,Z 52.000,A 180.000,B 0.000,C 180.000} C_DIS
LIN {X 11.852,Y 41.243,Z 52.000,A 180.000,B 0.000,C 180.000} C_DIS
LIN {X 11.852,Y 41.243,Z 57.000,A 180.000,B 0.000,C 180.000} C_DIS
LIN {X 30.690,Y 41.243,Z 57.000,A 180.000,B 0.000,C 180.000} C_DIS
LIN {X 30.694,Y 41.243,Z 52.000,A 180.000,B 0.000,C 180.000} C_DIS
LIN {X 42.306,Y 41.243,Z 52.000,A 180.000,B 0.000,C 180.000} C_DIS
LIN {X 42.306,Y 41.243,Z 57.000,A 180.000,B 0.000,C 180.000} C_DIS
LIN {X 45.221,Y 41.243,Z 57.000,A 180.000,B 0.000,C 180.000} C_DIS
LIN {X 45.221,Y 41.243,Z 62.000,A 180.000,B 0.000,C 180.000} C_DIS
LIN {X 71.941,Y 41.243,Z 62.000,A 180.000,B 0.000,C 180.000} C_DIS
LIN {X 71.941,Y 41.243,Z 70.721,A 180.000,B 0.000,C 180.000} C_DIS
LIN {X 71.952,Y 41.243,Z 70.769,A 180.000,B 0.000,C 180.000} C_DIS
LIN {X 71.991,Y 41.243,Z 70.813,A 180.000,B 0.000,C 180.000} C_DIS
LIN {X 72.066,Y 41.243,Z 70.850,A 180.000,B 0.000,C 180.000} C_DIS
LIN {X 72.198,Y 41.243,Z 70.876,A 180.000,B 0.000,C 180.000} C_DIS
LIN {X 72.419,Y 41.243,Z 70.882,A 180.000,B 0.000,C 180.000} C_DIS
LIN {X 72.656,Y 41.243,Z 70.866,A 180.000,B 0.000,C 180.000} C_DIS
LIN {X 73.082,Y 41.243,Z 70.808,A 180.000,B 0.000,C 180.000} C_DIS
LIN {X 73.686,Y 41.243,Z 70.690,A 180.000,B 0.000,C 180.000} C_DIS
LIN {X 74.507,Y 41.243,Z 70.522,A 180.000,B 0.000,C 180.000} C_DIS
LIN {X 75.576,Y 41.243,Z 70.315,A 180.000,B 0.000,C 180.000} C_DIS
LIN {X 75.732,Y 41.243,Z 70.355,A 180.000,B 0.000,C 180.000} C_DIS
LIN {X 76.197,Y 41.243,Z 70.503,A 180.000,B 0.000,C 180.000} C_DIS
LIN {X 76.647,Y 41.243,Z 70.667,A 180.000,B 0.000,C 180.000} C_DIS
LIN {X 77.162,Y 41.243,Z 70.884,A 180.000,B 0.000,C 180.000} C_DIS
LIN {X 77.681,Y 41.243,Z 71.126,A 180.000,B 0.000,C 180.000} C_DIS
LIN {X 78.240,Y 41.243,Z 71.417,A 180.000,B 0.000,C 180.000} C_DIS
LIN {X 78.838,Y 41.243,Z 71.754,A 180.000,B 0.000,C 180.000} C_DIS
LIN {X 79.473,Y 41.243,Z 72.141,A 180.000,B 0.000,C 180.000} C_DIS
LIN {X 80.184,Y 41.243,Z 72.607,A 180.000,B 0.000,C 180.000} C_DIS
LIN {X 80.942,Y 41.243,Z 73.150,A 180.000,B 0.000,C 180.000} C_DIS
LIN {X 81.670,Y 41.243,Z 73.716,A 180.000,B 0.000,C 180.000} C_DIS
LIN {X 82.439,Y 41.243,Z 74.361,A 180.000,B 0.000,C 180.000} C_DIS
LIN {X 87.717,Y 41.243,Z 74.364,A 180.000,B 0.000,C 180.000} C_DIS
LIN {X 93.028,Y 41.243,Z 72.155,A 180.000,B 0.000,C 180.000} C_DIS
LIN {X 93.028,Y 41.243,Z 70.198,A 180.000,B 0.000,C 180.000} C_DIS
LIN {X 93.517,Y 41.243,Z 70.191,A 180.000,B 0.000,C 180.000} C_DIS
LIN {X 94.357,Y 41.243,Z 70.170,A 180.000,B 0.000,C 180.000} C_DIS
LIN {X 94.854,Y 41.243,Z 70.142,A 180.000,B 0.000,C 180.000} C_DIS
LIN {X 95.707,Y 41.243,Z 70.076,A 180.000,B 0.000,C 180.000} C_DIS
LIN {X 96.193,Y 41.243,Z 70.015,A 180.000,B 0.000,C 180.000} C_DIS
LIN {X 96.777,Y 41.243,Z 69.930,A 180.000,B 0.000,C 180.000} C_DIS
LIN {X 97.547,Y 41.243,Z 69.769,A 180.000,B 0.000,C 180.000} C_DIS
LIN {X 98.278,Y 41.243,Z 69.563,A 180.000,B 0.000,C 180.000} C_DIS
LIN {X 98.952,Y 41.243,Z 69.315,A 180.000,B 0.000,C 180.000} C_DIS
LIN {X 99.571,Y 41.243,Z 69.029,A 180.000,B 0.000,C 180.000} C_DIS
LIN {X 100.100,Y 41.243,Z 68.733,A 180.000,B 0.000,C 180.000} C_DIS
LIN {X 100.628,Y 41.243,Z 68.379,A 180.000,B 0.000,C 180.000} C_DIS
LIN {X 101.075,Y 41.243,Z 68.023,A 180.000,B 0.000,C 180.000} C_DIS
LIN {X 101.489,Y 41.243,Z 67.630,A 180.000,B 0.000,C 180.000} C_DIS
LIN {X 101.878,Y 41.243,Z 67.201,A 180.000,B 0.000,C 180.000} C_DIS
LIN {X 102.206,Y 41.243,Z 66.769,A 180.000,B 0.000,C 180.000} C_DIS
LIN {X 102.497,Y 41.243,Z 66.303,A 180.000,B 0.000,C 180.000} C_DIS
LIN {X 102.744,Y 41.243,Z 65.821,A 180.000,B 0.000,C 180.000} C_DIS
LIN {X 102.948,Y 41.243,Z 65.329,A 180.000,B 0.000,C 180.000} C_DIS
LIN {X 103.106,Y 41.243,Z 64.829,A 180.000,B 0.000,C 180.000} C_DIS
LIN {X 103.221,Y 41.243,Z 64.320,A 180.000,B 0.000,C 180.000} C_DIS
LIN {X 103.292,Y 41.243,Z 63.804,A 180.000,B 0.000,C 180.000} C_DIS
LIN {X 103.316,Y 41.243,Z 63.319,A 180.000,B 0.000,C 180.000} C_DIS
LIN {X 103.319,Y 41.243,Z 62.000,A 180.000,B 0.000,C 180.000} C_DIS
LIN {X 109.779,Y 41.243,Z 62.000,A 180.000,B 0.000,C 180.000} C_DIS
LIN {X 109.779,Y 41.243,Z 57.000,A 180.000,B 0.000,C 180.000} C_DIS
LIN {X 112.690,Y 41.243,Z 57.000,A 180.000,B 0.000,C 180.000} C_DIS
LIN {X 112.694,Y 41.243,Z 52.000,A 180.000,B 0.000,C 180.000} C_DIS
LIN {X 124.306,Y 41.243,Z 52.000,A 180.000,B 0.000,C 180.000} C_DIS
LIN {X 124.306,Y 41.243,Z 57.000,A 180.000,B 0.000,C 180.000} C_DIS
LIN {X 143.148,Y 41.243,Z 57.000,A 180.000,B 0.000,C 180.000} C_DIS
LIN {X 143.148,Y 41.243,Z 52.000,A 180.000,B 0.000,C 180.000} C_DIS
LIN {X 152.500,Y 41.243,Z 52.000,A 180.000,B 0.000,C 180.000} C_DIS
LIN {X 152.500,Y 41.243,Z 45.000,A 180.000,B 0.000,C 180.000} C_DIS
LIN {X 155.010,Y 41.243,Z 45.000,A 180.000,B 0.000,C 180.000} C_DIS
; Link Move Starts
LIN {X 155.120,Y 41.243,Z 45.026,A 180.000,B 0.000,C 180.000} C_DIS
LIN {X 155.230,Y 41.243,Z 45.051,A 180.000,B 0.000,C 180.000} C_DIS
LIN {X 155.771,Y 41.556,Z 45.051,A 180.000,B 0.000,C 180.000} C_DIS
LIN {X 155.771,Y 42.181,Z 45.051,A 180.000,B 0.000,C 180.000} C_DIS
LIN {X 155.230,Y 42.493,Z 45.051,A 180.000,B 0.000,C 180.000} C_DIS
LIN {X 155.120,Y 42.493,Z 45.026,A 180.000,B 0.000,C 180.000} C_DIS
LIN {X 155.010,Y 42.493,Z 45.000,A 180.000,B 0.000,C 180.000} C_DIS
; Cutting Move Starts
LIN {X 152.500,Y 42.493,Z 45.000,A 180.000,B 0.000,C 180.000} C_DIS
LIN {X 152.500,Y 42.493,Z 52.000,A 180.000,B 0.000,C 180.000} C_DIS
LIN {X 143.824,Y 42.493,Z 52.000,A 180.000,B 0.000,C 180.000} C_DIS
LIN {X 143.822,Y 42.493,Z 57.000,A 180.000,B 0.000,C 180.000} C_DIS
LIN {X 123.002,Y 42.493,Z 57.000,A 180.000,B 0.000,C 180.000} C_DIS
LIN {X 123.002,Y 42.493,Z 52.000,A 180.000,B 0.000,C 180.000} C_DIS
LIN {X 113.998,Y 42.493,Z 52.000,A 180.000,B 0.000,C 180.000} C_DIS
LIN {X 113.998,Y 42.493,Z 57.000,A 180.000,B 0.000,C 180.000} C_DIS
LIN {X 111.029,Y 42.493,Z 57.000,A 180.000,B 0.000,C 180.000} C_DIS
LIN {X 111.029,Y 42.493,Z 62.000,A 180.000,B 0.000,C 180.000} C_DIS
LIN {X 103.948,Y 42.493,Z 62.000,A 180.000,B 0.000,C 180.000} C_DIS
LIN {X 103.945,Y 42.493,Z 63.322,A 180.000,B 0.000,C 180.000} C_DIS
LIN {X 103.924,Y 42.493,Z 63.795,A 180.000,B 0.000,C 180.000} C_DIS
LIN {X 103.854,Y 42.493,Z 64.333,A 180.000,B 0.000,C 180.000} C_DIS
LIN {X 103.744,Y 42.493,Z 64.847,A 180.000,B 0.000,C 180.000} C_DIS
LIN {X 103.599,Y 42.493,Z 65.333,A 180.000,B 0.000,C 180.000} C_DIS
LIN {X 103.407,Y 42.493,Z 65.828,A 180.000,B 0.000,C 180.000} C_DIS
LIN {X 103.179,Y 42.493,Z 66.303,A 180.000,B 0.000,C 180.000} C_DIS
LIN {X 102.899,Y 42.493,Z 66.779,A 180.000,B 0.000,C 180.000} C_DIS
LIN {X 102.597,Y 42.493,Z 67.206,A 180.000,B 0.000,C 180.000} C_DIS
LIN {X 102.240,Y 42.493,Z 67.631,A 180.000,B 0.000,C 180.000} C_DIS
LIN {X 101.854,Y 42.493,Z 68.026,A 180.000,B 0.000,C 180.000} C_DIS
LIN {X 101.433,Y 42.493,Z 68.396,A 180.000,B 0.000,C 180.000} C_DIS
LIN {X 100.975,Y 42.493,Z 68.733,A 180.000,B 0.000,C 180.000} C_DIS
LIN {X 100.476,Y 42.493,Z 69.045,A 180.000,B 0.000,C 180.000} C_DIS
LIN {X 99.958,Y 42.493,Z 69.317,A 180.000,B 0.000,C 180.000} C_DIS
LIN {X 99.386,Y 42.493,Z 69.563,A 180.000,B 0.000,C 180.000} C_DIS
LIN {X 98.792,Y 42.493,Z 69.768,A 180.000,B 0.000,C 180.000} C_DIS
LIN {X 98.158,Y 42.493,Z 69.937,A 180.000,B 0.000,C 180.000} C_DIS
LIN {X 97.470,Y 42.493,Z 70.071,A 180.000,B 0.000,C 180.000} C_DIS
LIN {X 96.708,Y 42.493,Z 70.169,A 180.000,B 0.000,C 180.000} C_DIS
LIN {X 95.851,Y 42.493,Z 70.227,A 180.000,B 0.000,C 180.000} C_DIS
LIN {X 94.673,Y 42.493,Z 70.247,A 180.000,B 0.000,C 180.000} C_DIS
LIN {X 93.449,Y 42.493,Z 70.247,A 180.000,B 0.000,C 180.000} C_DIS
LIN {X 93.449,Y 42.493,Z 72.155,A 180.000,B 0.000,C 180.000} C_DIS
LIN {X 88.139,Y 42.493,Z 74.364,A 180.000,B 0.000,C 180.000} C_DIS
LIN {X 82.861,Y 42.493,Z 74.361,A 180.000,B 0.000,C 180.000} C_DIS
LIN {X 82.091,Y 42.493,Z 73.716,A 180.000,B 0.000,C 180.000} C_DIS
LIN {X 81.363,Y 42.493,Z 73.150,A 180.000,B 0.000,C 180.000} C_DIS
LIN {X 80.606,Y 42.493,Z 72.607,A 180.000,B 0.000,C 180.000} C_DIS
LIN {X 79.920,Y 42.493,Z 72.157,A 180.000,B 0.000,C 180.000} C_DIS
LIN {X 79.252,Y 42.493,Z 71.760,A 180.000,B 0.000,C 180.000} C_DIS
LIN {X 78.598,Y 42.493,Z 71.411,A 180.000,B 0.000,C 180.000} C_DIS
LIN {X 77.949,Y 42.493,Z 71.101,A 180.000,B 0.000,C 180.000} C_DIS
LIN {X 77.332,Y 42.493,Z 70.843,A 180.000,B 0.000,C 180.000} C_DIS
LIN {X 76.712,Y 42.493,Z 70.622,A 180.000,B 0.000,C 180.000} C_DIS
LIN {X 76.088,Y 42.493,Z 70.435,A 180.000,B 0.000,C 180.000} C_DIS
LIN {X 76.005,Y 42.493,Z 70.416,A 180.000,B 0.000,C 180.000} C_DIS
LIN {X 75.616,Y 42.493,Z 70.520,A 180.000,B 0.000,C 180.000} C_DIS
LIN {X 74.960,Y 42.493,Z 70.726,A 180.000,B 0.000,C 180.000} C_DIS
LIN {X 74.287,Y 42.493,Z 70.968,A 180.000,B 0.000,C 180.000} C_DIS
LIN {X 73.589,Y 42.493,Z 71.247,A 180.000,B 0.000,C 180.000} C_DIS
LIN {X 72.859,Y 42.493,Z 71.560,A 180.000,B 0.000,C 180.000} C_DIS
LIN {X 72.049,Y 42.493,Z 71.926,A 180.000,B 0.000,C 180.000} C_DIS
LIN {X 70.786,Y 42.493,Z 72.499,A 180.000,B 0.000,C 180.000} C_DIS
LIN {X 70.124,Y 42.493,Z 72.783,A 180.000,B 0.000,C 180.000} C_DIS
LIN {X 69.524,Y 42.493,Z 73.007,A 180.000,B 0.000,C 180.000} C_DIS
LIN {X 69.165,Y 42.493,Z 73.116,A 180.000,B 0.000,C 180.000} C_DIS
LIN {X 68.884,Y 42.493,Z 73.175,A 180.000,B 0.000,C 180.000} C_DIS
LIN {X 68.702,Y 42.493,Z 73.194,A 180.000,B 0.000,C 180.000} C_DIS
LIN {X 68.533,Y 42.493,Z 73.189,A 180.000,B 0.000,C 180.000} C_DIS
LIN {X 68.410,Y 42.493,Z 73.158,A 180.000,B 0.000,C 180.000} C_DIS
LIN {X 68.330,Y 42.493,Z 73.112,A 180.000,B 0.000,C 180.000} C_DIS
LIN {X 68.276,Y 42.493,Z 73.051,A 180.000,B 0.000,C 180.000} C_DIS
LIN {X 68.244,Y 42.493,Z 72.970,A 180.000,B 0.000,C 180.000} C_DIS
LIN {X 68.236,Y 42.493,Z 72.895,A 180.000,B 0.000,C 180.000} C_DIS
LIN {X 68.236,Y 42.493,Z 62.000,A 180.000,B 0.000,C 180.000} C_DIS
LIN {X 43.971,Y 42.493,Z 62.000,A 180.000,B 0.000,C 180.000} C_DIS
LIN {X 43.971,Y 42.493,Z 57.000,A 180.000,B 0.000,C 180.000} C_DIS
LIN {X 41.002,Y 42.493,Z 57.000,A 180.000,B 0.000,C 180.000} C_DIS
LIN {X 41.002,Y 42.493,Z 52.000,A 180.000,B 0.000,C 180.000} C_DIS
LIN {X 31.998,Y 42.493,Z 52.000,A 180.000,B 0.000,C 180.000} C_DIS
LIN {X 31.998,Y 42.493,Z 57.000,A 180.000,B 0.000,C 180.000} C_DIS
LIN {X 11.176,Y 42.493,Z 57.000,A 180.000,B 0.000,C 180.000} C_DIS
LIN {X 11.176,Y 42.493,Z 52.000,A 180.000,B 0.000,C 180.000} C_DIS
LIN {X 2.500,Y 42.493,Z 52.000,A 180.000,B 0.000,C 180.000} C_DIS
LIN {X 2.500,Y 42.493,Z 45.000,A 180.000,B 0.000,C 180.000} C_DIS
LIN {X -0.010,Y 42.493,Z 45.000,A 180.000,B 0.000,C 180.000} C_DIS
; Link Move Starts
LIN {X -0.120,Y 42.493,Z 45.026,A 180.000,B 0.000,C 180.000} C_DIS
LIN {X -0.230,Y 42.493,Z 45.051,A 180.000,B 0.000,C 180.000} C_DIS
LIN {X -0.771,Y 42.806,Z 45.051,A 180.000,B 0.000,C 180.000} C_DIS
LIN {X -0.771,Y 43.431,Z 45.051,A 180.000,B 0.000,C 180.000} C_DIS
LIN {X -0.230,Y 43.743,Z 45.051,A 180.000,B 0.000,C 180.000} C_DIS
LIN {X -0.120,Y 43.743,Z 45.026,A 180.000,B 0.000,C 180.000} C_DIS
LIN {X -0.010,Y 43.743,Z 45.000,A 180.000,B 0.000,C 180.000} C_DIS
; Cutting Move Starts
LIN {X 2.500,Y 43.743,Z 45.000,A 180.000,B 0.000,C 180.000} C_DIS
LIN {X 2.500,Y 43.743,Z 52.000,A 180.000,B 0.000,C 180.000} C_DIS
LIN {X 10.528,Y 43.743,Z 52.000,A 180.000,B 0.000,C 180.000} C_DIS
LIN {X 10.528,Y 43.743,Z 57.000,A 180.000,B 0.000,C 180.000} C_DIS
LIN {X 34.562,Y 43.743,Z 57.000,A 180.000,B 0.000,C 180.000} C_DIS
LIN {X 34.566,Y 43.743,Z 52.000,A 180.000,B 0.000,C 180.000} C_DIS
LIN {X 38.434,Y 43.743,Z 52.000,A 180.000,B 0.000,C 180.000} C_DIS
LIN {X 38.434,Y 43.743,Z 57.000,A 180.000,B 0.000,C 180.000} C_DIS
LIN {X 42.719,Y 43.743,Z 57.000,A 180.000,B 0.000,C 180.000} C_DIS
LIN {X 42.721,Y 43.743,Z 62.000,A 180.000,B 0.000,C 180.000} C_DIS
LIN {X 64.531,Y 43.743,Z 62.000,A 180.000,B 0.000,C 180.000} C_DIS
LIN {X 64.534,Y 43.743,Z 76.129,A 180.000,B 0.000,C 180.000} C_DIS
LIN {X 64.557,Y 43.743,Z 76.229,A 180.000,B 0.000,C 180.000} C_DIS
LIN {X 64.602,Y 43.743,Z 76.307,A 180.000,B 0.000,C 180.000} C_DIS
LIN {X 64.670,Y 43.743,Z 76.366,A 180.000,B 0.000,C 180.000} C_DIS
LIN {X 64.761,Y 43.743,Z 76.406,A 180.000,B 0.000,C 180.000} C_DIS
LIN {X 64.883,Y 43.743,Z 76.427,A 180.000,B 0.000,C 180.000} C_DIS
LIN {X 65.060,Y 43.743,Z 76.423,A 180.000,B 0.000,C 180.000} C_DIS
LIN {X 65.276,Y 43.743,Z 76.385,A 180.000,B 0.000,C 180.000} C_DIS
LIN {X 65.561,Y 43.743,Z 76.303,A 180.000,B 0.000,C 180.000} C_DIS
LIN {X 65.915,Y 43.743,Z 76.168,A 180.000,B 0.000,C 180.000} C_DIS
LIN {X 66.364,Y 43.743,Z 75.962,A 180.000,B 0.000,C 180.000} C_DIS
LIN {X 66.896,Y 43.743,Z 75.686,A 180.000,B 0.000,C 180.000} C_DIS
LIN {X 67.523,Y 43.743,Z 75.324,A 180.000,B 0.000,C 180.000} C_DIS
LIN {X 68.547,Y 43.743,Z 74.690,A 180.000,B 0.000,C 180.000} C_DIS
LIN {X 70.598,Y 43.743,Z 73.334,A 180.000,B 0.000,C 180.000} C_DIS
LIN {X 71.609,Y 43.743,Z 72.680,A 180.000,B 0.000,C 180.000} C_DIS
LIN {X 72.240,Y 43.743,Z 72.284,A 180.000,B 0.000,C 180.000} C_DIS
LIN {X 72.876,Y 43.743,Z 71.907,A 180.000,B 0.000,C 180.000} C_DIS
LIN {X 73.502,Y 43.743,Z 71.565,A 180.000,B 0.000,C 180.000} C_DIS
LIN {X 74.124,Y 43.743,Z 71.257,A 180.000,B 0.000,C 180.000} C_DIS
LIN {X 74.756,Y 43.743,Z 70.978,A 180.000,B 0.000,C 180.000} C_DIS
LIN {X 75.384,Y 43.743,Z 70.735,A 180.000,B 0.000,C 180.000} C_DIS
LIN {X 76.008,Y 43.743,Z 70.531,A 180.000,B 0.000,C 180.000} C_DIS
LIN {X 76.429,Y 43.743,Z 70.415,A 180.000,B 0.000,C 180.000} C_DIS
LIN {X 76.511,Y 43.743,Z 70.435,A 180.000,B 0.000,C 180.000} C_DIS
LIN {X 77.134,Y 43.743,Z 70.622,A 180.000,B 0.000,C 180.000} C_DIS
LIN {X 77.753,Y 43.743,Z 70.843,A 180.000,B 0.000,C 180.000} C_DIS
LIN {X 78.371,Y 43.743,Z 71.101,A 180.000,B 0.000,C 180.000} C_DIS
LIN {X 79.020,Y 43.743,Z 71.411,A 180.000,B 0.000,C 180.000} C_DIS
LIN {X 79.674,Y 43.743,Z 71.760,A 180.000,B 0.000,C 180.000} C_DIS
LIN {X 80.341,Y 43.743,Z 72.157,A 180.000,B 0.000,C 180.000} C_DIS
LIN {X 81.027,Y 43.743,Z 72.607,A 180.000,B 0.000,C 180.000} C_DIS
LIN {X 81.785,Y 43.743,Z 73.150,A 180.000,B 0.000,C 180.000} C_DIS
LIN {X 82.513,Y 43.743,Z 73.716,A 180.000,B 0.000,C 180.000} C_DIS
LIN {X 83.283,Y 43.743,Z 74.361,A 180.000,B 0.000,C 180.000} C_DIS
LIN {X 88.561,Y 43.743,Z 74.364,A 180.000,B 0.000,C 180.000} C_DIS
LIN {X 93.871,Y 43.743,Z 72.155,A 180.000,B 0.000,C 180.000} C_DIS
LIN {X 93.871,Y 43.743,Z 70.247,A 180.000,B 0.000,C 180.000} C_DIS
LIN {X 96.444,Y 43.743,Z 70.247,A 180.000,B 0.000,C 180.000} C_DIS
LIN {X 97.193,Y 43.743,Z 70.227,A 180.000,B 0.000,C 180.000} C_DIS
LIN {X 97.847,Y 43.743,Z 70.169,A 180.000,B 0.000,C 180.000} C_DIS
LIN {X 98.450,Y 43.743,Z 70.075,A 180.000,B 0.000,C 180.000} C_DIS
LIN {X 99.021,Y 43.743,Z 69.945,A 180.000,B 0.000,C 180.000} C_DIS
LIN {X 99.599,Y 43.743,Z 69.771,A 180.000,B 0.000,C 180.000} C_DIS
LIN {X 100.123,Y 43.743,Z 69.570,A 180.000,B 0.000,C 180.000} C_DIS
LIN {X 100.653,Y 43.743,Z 69.320,A 180.000,B 0.000,C 180.000} C_DIS
LIN {X 101.139,Y 43.743,Z 69.043,A 180.000,B 0.000,C 180.000} C_DIS
LIN {X 101.582,Y 43.743,Z 68.746,A 180.000,B 0.000,C 180.000} C_DIS
LIN {X 102.027,Y 43.743,Z 68.394,A 180.000,B 0.000,C 180.000} C_DIS
LIN {X 102.423,Y 43.743,Z 68.025,A 180.000,B 0.000,C 180.000} C_DIS
LIN {X 102.788,Y 43.743,Z 67.630,A 180.000,B 0.000,C 180.000} C_DIS
LIN {X 103.121,Y 43.743,Z 67.210,A 180.000,B 0.000,C 180.000} C_DIS
LIN {X 103.408,Y 43.743,Z 66.785,A 180.000,B 0.000,C 180.000} C_DIS
LIN {X 103.671,Y 43.743,Z 66.324,A 180.000,B 0.000,C 180.000} C_DIS
LIN {X 103.903,Y 43.743,Z 65.825,A 180.000,B 0.000,C 180.000} C_DIS
LIN {X 104.084,Y 43.743,Z 65.334,A 180.000,B 0.000,C 180.000} C_DIS
LIN {X 104.223,Y 43.743,Z 64.846,A 180.000,B 0.000,C 180.000} C_DIS
LIN {X 104.328,Y 43.743,Z 64.331,A 180.000,B 0.000,C 180.000} C_DIS
LIN {X 104.393,Y 43.743,Z 63.807,A 180.000,B 0.000,C 180.000} C_DIS
LIN {X 104.416,Y 43.743,Z 63.301,A 180.000,B 0.000,C 180.000} C_DIS
LIN {X 104.418,Y 43.743,Z 62.000,A 180.000,B 0.000,C 180.000} C_DIS
LIN {X 112.279,Y 43.743,Z 62.000,A 180.000,B 0.000,C 180.000} C_DIS
LIN {X 112.279,Y 43.743,Z 57.000,A 180.000,B 0.000,C 180.000} C_DIS
LIN {X 116.562,Y 43.743,Z 57.000,A 180.000,B 0.000,C 180.000} C_DIS
LIN {X 116.566,Y 43.743,Z 52.000,A 180.000,B 0.000,C 180.000} C_DIS
LIN {X 120.434,Y 43.743,Z 52.000,A 180.000,B 0.000,C 180.000} C_DIS
LIN {X 120.434,Y 43.743,Z 57.000,A 180.000,B 0.000,C 180.000} C_DIS
LIN {X 144.472,Y 43.743,Z 57.000,A 180.000,B 0.000,C 180.000} C_DIS
LIN {X 144.472,Y 43.743,Z 52.000,A 180.000,B 0.000,C 180.000} C_DIS
LIN {X 152.500,Y 43.743,Z 52.000,A 180.000,B 0.000,C 180.000} C_DIS
LIN {X 152.500,Y 43.743,Z 45.000,A 180.000,B 0.000,C 180.000} C_DIS
LIN {X 155.010,Y 43.743,Z 45.000,A 180.000,B 0.000,C 180.000} C_DIS
; Link Move Starts
LIN {X 155.120,Y 43.743,Z 45.026,A 180.000,B 0.000,C 180.000} C_DIS
LIN {X 155.230,Y 43.743,Z 45.051,A 180.000,B 0.000,C 180.000} C_DIS
LIN {X 155.771,Y 44.056,Z 45.051,A 180.000,B 0.000,C 180.000} C_DIS
LIN {X 155.771,Y 44.681,Z 45.051,A 180.000,B 0.000,C 180.000} C_DIS
LIN {X 155.230,Y 44.993,Z 45.051,A 180.000,B 0.000,C 180.000} C_DIS
LIN {X 155.120,Y 44.993,Z 45.026,A 180.000,B 0.000,C 180.000} C_DIS
LIN {X 155.010,Y 44.993,Z 45.000,A 180.000,B 0.000,C 180.000} C_DIS
; Cutting Move Starts
LIN {X 152.500,Y 44.993,Z 45.000,A 180.000,B 0.000,C 180.000} C_DIS
LIN {X 152.500,Y 44.993,Z 52.000,A 180.000,B 0.000,C 180.000} C_DIS
LIN {X 145.087,Y 44.993,Z 52.000,A 180.000,B 0.000,C 180.000} C_DIS
LIN {X 145.087,Y 44.993,Z 57.000,A 180.000,B 0.000,C 180.000} C_DIS
LIN {X 113.529,Y 44.993,Z 57.000,A 180.000,B 0.000,C 180.000} C_DIS
LIN {X 113.529,Y 44.993,Z 62.000,A 180.000,B 0.000,C 180.000} C_DIS
LIN {X 104.746,Y 44.993,Z 62.000,A 180.000,B 0.000,C 180.000} C_DIS
LIN {X 104.743,Y 44.993,Z 63.321,A 180.000,B 0.000,C 180.000} C_DIS
LIN {X 104.719,Y 44.993,Z 63.829,A 180.000,B 0.000,C 180.000} C_DIS
LIN {X 104.654,Y 44.993,Z 64.350,A 180.000,B 0.000,C 180.000} C_DIS
LIN {X 104.550,Y 44.993,Z 64.863,A 180.000,B 0.000,C 180.000} C_DIS
LIN {X 104.419,Y 44.993,Z 65.334,A 180.000,B 0.000,C 180.000} C_DIS
LIN {X 104.240,Y 44.993,Z 65.825,A 180.000,B 0.000,C 180.000} C_DIS
LIN {X 104.021,Y 44.993,Z 66.309,A 180.000,B 0.000,C 180.000} C_DIS
LIN {X 103.770,Y 44.993,Z 66.767,A 180.000,B 0.000,C 180.000} C_DIS
LIN {X 103.482,Y 44.993,Z 67.210,A 180.000,B 0.000,C 180.000} C_DIS
LIN {X 103.161,Y 44.993,Z 67.631,A 180.000,B 0.000,C 180.000} C_DIS
LIN {X 102.811,Y 44.993,Z 68.025,A 180.000,B 0.000,C 180.000} C_DIS
LIN {X 102.426,Y 44.993,Z 68.396,A 180.000,B 0.000,C 180.000} C_DIS
LIN {X 102.012,Y 44.993,Z 68.740,A 180.000,B 0.000,C 180.000} C_DIS
LIN {X 101.561,Y 44.993,Z 69.056,A 180.000,B 0.000,C 180.000} C_DIS
LIN {X 101.121,Y 44.993,Z 69.319,A 180.000,B 0.000,C 180.000} C_DIS
LIN {X 100.637,Y 44.993,Z 69.562,A 180.000,B 0.000,C 180.000} C_DIS
LIN {X 100.129,Y 44.993,Z 69.772,A 180.000,B 0.000,C 180.000} C_DIS
LIN {X 99.609,Y 44.993,Z 69.942,A 180.000,B 0.000,C 180.000} C_DIS
LIN {X 99.073,Y 44.993,Z 70.075,A 180.000,B 0.000,C 180.000} C_DIS
LIN {X 98.503,Y 44.993,Z 70.173,A 180.000,B 0.000,C 180.000} C_DIS
LIN {X 97.961,Y 44.993,Z 70.228,A 180.000,B 0.000,C 180.000} C_DIS
LIN {X 97.348,Y 44.993,Z 70.247,A 180.000,B 0.000,C 180.000} C_DIS
LIN {X 94.293,Y 44.993,Z 70.247,A 180.000,B 0.000,C 180.000} C_DIS
LIN {X 94.292,Y 44.993,Z 72.155,A 180.000,B 0.000,C 180.000} C_DIS
LIN {X 88.982,Y 44.993,Z 74.364,A 180.000,B 0.000,C 180.000} C_DIS
LIN {X 83.704,Y 44.993,Z 74.361,A 180.000,B 0.000,C 180.000} C_DIS
LIN {X 82.935,Y 44.993,Z 73.716,A 180.000,B 0.000,C 180.000} C_DIS
LIN {X 82.207,Y 44.993,Z 73.150,A 180.000,B 0.000,C 180.000} C_DIS
LIN {X 81.449,Y 44.993,Z 72.607,A 180.000,B 0.000,C 180.000} C_DIS
LIN {X 80.763,Y 44.993,Z 72.157,A 180.000,B 0.000,C 180.000} C_DIS
LIN {X 80.096,Y 44.993,Z 71.760,A 180.000,B 0.000,C 180.000} C_DIS
LIN {X 79.442,Y 44.993,Z 71.411,A 180.000,B 0.000,C 180.000} C_DIS
LIN {X 78.793,Y 44.993,Z 71.101,A 180.000,B 0.000,C 180.000} C_DIS
LIN {X 78.175,Y 44.993,Z 70.843,A 180.000,B 0.000,C 180.000} C_DIS
LIN {X 77.555,Y 44.993,Z 70.622,A 180.000,B 0.000,C 180.000} C_DIS
LIN {X 76.932,Y 44.993,Z 70.435,A 180.000,B 0.000,C 180.000} C_DIS
LIN {X 76.851,Y 44.993,Z 70.415,A 180.000,B 0.000,C 180.000} C_DIS
LIN {X 76.429,Y 44.993,Z 70.531,A 180.000,B 0.000,C 180.000} C_DIS
LIN {X 75.806,Y 44.993,Z 70.735,A 180.000,B 0.000,C 180.000} C_DIS
LIN {X 75.178,Y 44.993,Z 70.978,A 180.000,B 0.000,C 180.000} C_DIS
LIN {X 74.545,Y 44.993,Z 71.257,A 180.000,B 0.000,C 180.000} C_DIS
LIN {X 73.924,Y 44.993,Z 71.565,A 180.000,B 0.000,C 180.000} C_DIS
LIN {X 73.298,Y 44.993,Z 71.907,A 180.000,B 0.000,C 180.000} C_DIS
LIN {X 72.670,Y 44.993,Z 72.279,A 180.000,B 0.000,C 180.000} C_DIS
LIN {X 72.031,Y 44.993,Z 72.687,A 180.000,B 0.000,C 180.000} C_DIS
LIN {X 71.352,Y 44.993,Z 73.149,A 180.000,B 0.000,C 180.000} C_DIS
LIN {X 70.454,Y 44.993,Z 73.798,A 180.000,B 0.000,C 180.000} C_DIS
LIN {X 69.625,Y 44.993,Z 74.436,A 180.000,B 0.000,C 180.000} C_DIS
LIN {X 68.443,Y 44.993,Z 75.377,A 180.000,B 0.000,C 180.000} C_DIS
LIN {X 67.378,Y 44.993,Z 76.220,A 180.000,B 0.000,C 180.000} C_DIS
LIN {X 66.416,Y 44.993,Z 76.949,A 180.000,B 0.000,C 180.000} C_DIS
LIN {X 65.516,Y 44.993,Z 77.597,A 180.000,B 0.000,C 180.000} C_DIS
LIN {X 64.926,Y 44.993,Z 77.999,A 180.000,B 0.000,C 180.000} C_DIS
LIN {X 64.152,Y 44.993,Z 78.483,A 180.000,B 0.000,C 180.000} C_DIS
LIN {X 63.516,Y 44.993,Z 78.852,A 180.000,B 0.000,C 180.000} C_DIS
LIN {X 62.919,Y 44.993,Z 79.157,A 180.000,B 0.000,C 180.000} C_DIS
LIN {X 62.518,Y 44.993,Z 79.339,A 180.000,B 0.000,C 180.000} C_DIS
LIN {X 62.083,Y 44.993,Z 79.508,A 180.000,B 0.000,C 180.000} C_DIS
LIN {X 61.739,Y 44.993,Z 79.615,A 180.000,B 0.000,C 180.000} C_DIS
LIN {X 61.474,Y 44.993,Z 79.673,A 180.000,B 0.000,C 180.000} C_DIS
LIN {X 61.282,Y 44.993,Z 79.694,A 180.000,B 0.000,C 180.000} C_DIS
LIN {X 61.122,Y 44.993,Z 79.688,A 180.000,B 0.000,C 180.000} C_DIS
LIN {X 61.008,Y 44.993,Z 79.659,A 180.000,B 0.000,C 180.000} C_DIS
LIN {X 60.925,Y 44.993,Z 79.612,A 180.000,B 0.000,C 180.000} C_DIS
LIN {X 60.869,Y 44.993,Z 79.549,A 180.000,B 0.000,C 180.000} C_DIS
LIN {X 60.836,Y 44.993,Z 79.467,A 180.000,B 0.000,C 180.000} C_DIS
LIN {X 60.826,Y 44.993,Z 79.378,A 180.000,B 0.000,C 180.000} C_DIS
LIN {X 60.826,Y 44.993,Z 62.000,A 180.000,B 0.000,C 180.000} C_DIS
LIN {X 41.471,Y 44.993,Z 62.000,A 180.000,B 0.000,C 180.000} C_DIS
LIN {X 41.471,Y 44.993,Z 57.000,A 180.000,B 0.000,C 180.000} C_DIS
LIN {X 9.913,Y 44.993,Z 57.000,A 180.000,B 0.000,C 180.000} C_DIS
LIN {X 9.913,Y 44.993,Z 52.000,A 180.000,B 0.000,C 180.000} C_DIS
LIN {X 2.500,Y 44.993,Z 52.000,A 180.000,B 0.000,C 180.000} C_DIS
LIN {X 2.500,Y 44.993,Z 45.000,A 180.000,B 0.000,C 180.000} C_DIS
LIN {X -0.010,Y 44.993,Z 45.000,A 180.000,B 0.000,C 180.000} C_DIS
; Link Move Starts
LIN {X -0.120,Y 44.993,Z 45.026,A 180.000,B 0.000,C 180.000} C_DIS
LIN {X -0.230,Y 44.993,Z 45.051,A 180.000,B 0.000,C 180.000} C_DIS
LIN {X -0.771,Y 45.306,Z 45.051,A 180.000,B 0.000,C 180.000} C_DIS
LIN {X -0.771,Y 45.931,Z 45.051,A 180.000,B 0.000,C 180.000} C_DIS
LIN {X -0.230,Y 46.243,Z 45.051,A 180.000,B 0.000,C 180.000} C_DIS
LIN {X -0.120,Y 46.243,Z 45.026,A 180.000,B 0.000,C 180.000} C_DIS
LIN {X -0.010,Y 46.243,Z 45.000,A 180.000,B 0.000,C 180.000} C_DIS
; Cutting Move Starts
LIN {X 2.500,Y 46.243,Z 45.000,A 180.000,B 0.000,C 180.000} C_DIS
LIN {X 2.500,Y 46.243,Z 52.000,A 180.000,B 0.000,C 180.000} C_DIS
LIN {X 9.329,Y 46.243,Z 52.000,A 180.000,B 0.000,C 180.000} C_DIS
LIN {X 9.329,Y 46.243,Z 57.000,A 180.000,B 0.000,C 180.000} C_DIS
LIN {X 40.221,Y 46.243,Z 57.000,A 180.000,B 0.000,C 180.000} C_DIS
LIN {X 40.221,Y 46.243,Z 62.000,A 180.000,B 0.000,C 180.000} C_DIS
LIN {X 57.121,Y 46.243,Z 62.000,A 180.000,B 0.000,C 180.000} C_DIS
LIN {X 57.122,Y 46.243,Z 81.927,A 180.000,B 0.000,C 180.000} C_DIS
LIN {X 57.135,Y 46.243,Z 81.976,A 180.000,B 0.000,C 180.000} C_DIS
LIN {X 57.173,Y 46.243,Z 82.024,A 180.000,B 0.000,C 180.000} C_DIS
LIN {X 57.246,Y 46.243,Z 82.065,A 180.000,B 0.000,C 180.000} C_DIS
LIN {X 57.364,Y 46.243,Z 82.094,A 180.000,B 0.000,C 180.000} C_DIS
LIN {X 57.544,Y 46.243,Z 82.104,A 180.000,B 0.000,C 180.000} C_DIS
LIN {X 57.818,Y 46.243,Z 82.086,A 180.000,B 0.000,C 180.000} C_DIS
LIN {X 58.190,Y 46.243,Z 82.029,A 180.000,B 0.000,C 180.000} C_DIS
LIN {X 58.691,Y 46.243,Z 81.919,A 180.000,B 0.000,C 180.000} C_DIS
LIN {X 59.066,Y 46.243,Z 81.814,A 180.000,B 0.000,C 180.000} C_DIS
LIN {X 59.766,Y 46.243,Z 81.585,A 180.000,B 0.000,C 180.000} C_DIS
LIN {X 60.542,Y 46.243,Z 81.275,A 180.000,B 0.000,C 180.000} C_DIS
LIN {X 61.274,Y 46.243,Z 80.935,A 180.000,B 0.000,C 180.000} C_DIS
LIN {X 61.967,Y 46.243,Z 80.571,A 180.000,B 0.000,C 180.000} C_DIS
LIN {X 62.623,Y 46.243,Z 80.191,A 180.000,B 0.000,C 180.000} C_DIS
LIN {X 63.250,Y 46.243,Z 79.794,A 180.000,B 0.000,C 180.000} C_DIS
LIN {X 63.866,Y 46.243,Z 79.374,A 180.000,B 0.000,C 180.000} C_DIS
LIN {X 64.567,Y 46.243,Z 78.863,A 180.000,B 0.000,C 180.000} C_DIS
LIN {X 65.687,Y 46.243,Z 77.982,A 180.000,B 0.000,C 180.000} C_DIS
LIN {X 68.904,Y 46.243,Z 75.345,A 180.000,B 0.000,C 180.000} C_DIS
LIN {X 70.046,Y 46.243,Z 74.436,A 180.000,B 0.000,C 180.000} C_DIS
LIN {X 70.875,Y 46.243,Z 73.798,A 180.000,B 0.000,C 180.000} C_DIS
LIN {X 71.773,Y 46.243,Z 73.149,A 180.000,B 0.000,C 180.000} C_DIS
LIN {X 72.453,Y 46.243,Z 72.687,A 180.000,B 0.000,C 180.000} C_DIS
LIN {X 73.092,Y 46.243,Z 72.279,A 180.000,B 0.000,C 180.000} C_DIS
LIN {X 73.720,Y 46.243,Z 71.907,A 180.000,B 0.000,C 180.000} C_DIS
LIN {X 74.345,Y 46.243,Z 71.565,A 180.000,B 0.000,C 180.000} C_DIS
LIN {X 74.967,Y 46.243,Z 71.257,A 180.000,B 0.000,C 180.000} C_DIS
LIN {X 75.599,Y 46.243,Z 70.978,A 180.000,B 0.000,C 180.000} C_DIS
LIN {X 76.228,Y 46.243,Z 70.735,A 180.000,B 0.000,C 180.000} C_DIS
LIN {X 76.851,Y 46.243,Z 70.531,A 180.000,B 0.000,C 180.000} C_DIS
LIN {X 77.272,Y 46.243,Z 70.415,A 180.000,B 0.000,C 180.000} C_DIS
LIN {X 77.354,Y 46.243,Z 70.435,A 180.000,B 0.000,C 180.000} C_DIS
LIN {X 77.977,Y 46.243,Z 70.622,A 180.000,B 0.000,C 180.000} C_DIS
LIN {X 78.597,Y 46.243,Z 70.843,A 180.000,B 0.000,C 180.000} C_DIS
LIN {X 79.214,Y 46.243,Z 71.101,A 180.000,B 0.000,C 180.000} C_DIS
LIN {X 79.863,Y 46.243,Z 71.411,A 180.000,B 0.000,C 180.000} C_DIS
LIN {X 80.517,Y 46.243,Z 71.760,A 180.000,B 0.000,C 180.000} C_DIS
LIN {X 81.185,Y 46.243,Z 72.157,A 180.000,B 0.000,C 180.000} C_DIS
LIN {X 81.871,Y 46.243,Z 72.607,A 180.000,B 0.000,C 180.000} C_DIS
LIN {X 82.628,Y 46.243,Z 73.150,A 180.000,B 0.000,C 180.000} C_DIS
LIN {X 83.356,Y 46.243,Z 73.716,A 180.000,B 0.000,C 180.000} C_DIS
LIN {X 84.126,Y 46.243,Z 74.361,A 180.000,B 0.000,C 180.000} C_DIS
LIN {X 89.404,Y 46.243,Z 74.364,A 180.000,B 0.000,C 180.000} C_DIS
LIN {X 94.714,Y 46.243,Z 72.155,A 180.000,B 0.000,C 180.000} C_DIS
LIN {X 94.714,Y 46.243,Z 70.247,A 180.000,B 0.000,C 180.000} C_DIS
LIN {X 97.805,Y 46.243,Z 70.247,A 180.000,B 0.000,C 180.000} C_DIS
LIN {X 98.369,Y 46.243,Z 70.228,A 180.000,B 0.000,C 180.000} C_DIS
LIN {X 98.879,Y 46.243,Z 70.173,A 180.000,B 0.000,C 180.000} C_DIS
LIN {X 99.417,Y 46.243,Z 70.076,A 180.000,B 0.000,C 180.000} C_DIS
LIN {X 99.928,Y 46.243,Z 69.943,A 180.000,B 0.000,C 180.000} C_DIS
LIN {X 100.428,Y 46.243,Z 69.772,A 180.000,B 0.000,C 180.000} C_DIS
LIN {X 100.923,Y 46.243,Z 69.562,A 180.000,B 0.000,C 180.000} C_DIS
LIN {X 101.367,Y 46.243,Z 69.332,A 180.000,B 0.000,C 180.000} C_DIS
LIN {X 101.817,Y 46.243,Z 69.056,A 180.000,B 0.000,C 180.000} C_DIS
LIN {X 102.262,Y 46.243,Z 68.735,A 180.000,B 0.000,C 180.000} C_DIS
LIN {X 102.661,Y 46.243,Z 68.396,A 180.000,B 0.000,C 180.000} C_DIS
LIN {X 103.037,Y 46.243,Z 68.025,A 180.000,B 0.000,C 180.000} C_DIS
LIN {X 103.380,Y 46.243,Z 67.631,A 180.000,B 0.000,C 180.000} C_DIS
LIN {X 103.695,Y 46.243,Z 67.209,A 180.000,B 0.000,C 180.000} C_DIS
LIN {X 103.974,Y 46.243,Z 66.771,A 180.000,B 0.000,C 180.000} C_DIS
LIN {X 104.224,Y 46.243,Z 66.304,A 180.000,B 0.000,C 180.000} C_DIS
LIN {X 104.436,Y 46.243,Z 65.825,A 180.000,B 0.000,C 180.000} C_DIS
LIN {X 104.611,Y 46.243,Z 65.333,A 180.000,B 0.000,C 180.000} C_DIS
LIN {X 104.744,Y 46.243,Z 64.845,A 180.000,B 0.000,C 180.000} C_DIS
LIN {X 104.846,Y 46.243,Z 64.329,A 180.000,B 0.000,C 180.000} C_DIS
LIN {X 104.907,Y 46.243,Z 63.815,A 180.000,B 0.000,C 180.000} C_DIS
LIN {X 104.929,Y 46.243,Z 63.313,A 180.000,B 0.000,C 180.000} C_DIS
LIN {X 104.932,Y 46.243,Z 62.000,A 180.000,B 0.000,C 180.000} C_DIS
LIN {X 114.779,Y 46.243,Z 62.000,A 180.000,B 0.000,C 180.000} C_DIS
LIN {X 114.779,Y 46.243,Z 57.000,A 180.000,B 0.000,C 180.000} C_DIS
LIN {X 145.671,Y 46.243,Z 57.000,A 180.000,B 0.000,C 180.000} C_DIS
LIN {X 145.671,Y 46.243,Z 52.000,A 180.000,B 0.000,C 180.000} C_DIS
LIN {X 152.500,Y 46.243,Z 52.000,A 180.000,B 0.000,C 180.000} C_DIS
LIN {X 152.500,Y 46.243,Z 45.000,A 180.000,B 0.000,C 180.000} C_DIS
LIN {X 155.010,Y 46.243,Z 45.000,A 180.000,B 0.000,C 180.000} C_DIS
; Link Move Starts
LIN {X 155.120,Y 46.243,Z 45.026,A 180.000,B 0.000,C 180.000} C_DIS
LIN {X 155.230,Y 46.243,Z 45.051,A 180.000,B 0.000,C 180.000} C_DIS
LIN {X 155.771,Y 46.555,Z 45.051,A 180.000,B 0.000,C 180.000} C_DIS
LIN {X 155.771,Y 47.180,Z 45.051,A 180.000,B 0.000,C 180.000} C_DIS
LIN {X 155.230,Y 47.493,Z 45.051,A 180.000,B 0.000,C 180.000} C_DIS
LIN {X 155.120,Y 47.493,Z 45.026,A 180.000,B 0.000,C 180.000} C_DIS
LIN {X 155.010,Y 47.493,Z 45.000,A 180.000,B 0.000,C 180.000} C_DIS
; Cutting Move Starts
LIN {X 152.500,Y 47.493,Z 45.000,A 180.000,B 0.000,C 180.000} C_DIS
LIN {X 152.500,Y 47.493,Z 52.000,A 180.000,B 0.000,C 180.000} C_DIS
LIN {X 146.230,Y 47.493,Z 52.000,A 180.000,B 0.000,C 180.000} C_DIS
LIN {X 146.230,Y 47.493,Z 57.000,A 180.000,B 0.000,C 180.000} C_DIS
LIN {X 116.028,Y 47.493,Z 57.000,A 180.000,B 0.000,C 180.000} C_DIS
LIN {X 116.028,Y 47.493,Z 62.000,A 180.000,B 0.000,C 180.000} C_DIS
LIN {X 104.998,Y 47.493,Z 62.000,A 180.000,B 0.000,C 180.000} C_DIS
LIN {X 104.994,Y 47.493,Z 63.354,A 180.000,B 0.000,C 180.000} C_DIS
LIN {X 104.975,Y 47.493,Z 63.801,A 180.000,B 0.000,C 180.000} C_DIS
LIN {X 104.911,Y 47.493,Z 64.333,A 180.000,B 0.000,C 180.000} C_DIS
LIN {X 104.812,Y 47.493,Z 64.843,A 180.000,B 0.000,C 180.000} C_DIS
LIN {X 104.680,Y 47.493,Z 65.330,A 180.000,B 0.000,C 180.000} C_DIS
LIN {X 104.505,Y 47.493,Z 65.824,A 180.000,B 0.000,C 180.000} C_DIS
LIN {X 104.293,Y 47.493,Z 66.305,A 180.000,B 0.000,C 180.000} C_DIS
LIN {X 104.047,Y 47.493,Z 66.768,A 180.000,B 0.000,C 180.000} C_DIS
LIN {X 103.765,Y 47.493,Z 67.212,A 180.000,B 0.000,C 180.000} C_DIS
LIN {X 103.454,Y 47.493,Z 67.631,A 180.000,B 0.000,C 180.000} C_DIS
LIN {X 103.111,Y 47.493,Z 68.026,A 180.000,B 0.000,C 180.000} C_DIS
LIN {X 102.740,Y 47.493,Z 68.395,A 180.000,B 0.000,C 180.000} C_DIS
LIN {X 102.342,Y 47.493,Z 68.735,A 180.000,B 0.000,C 180.000} C_DIS
LIN {X 101.919,Y 47.493,Z 69.045,A 180.000,B 0.000,C 180.000} C_DIS
LIN {X 101.475,Y 47.493,Z 69.321,A 180.000,B 0.000,C 180.000} C_DIS
LIN {X 101.014,Y 47.493,Z 69.563,A 180.000,B 0.000,C 180.000} C_DIS
LIN {X 100.533,Y 47.493,Z 69.771,A 180.000,B 0.000,C 180.000} C_DIS
LIN {X 100.033,Y 47.493,Z 69.944,A 180.000,B 0.000,C 180.000} C_DIS
LIN {X 99.511,Y 47.493,Z 70.080,A 180.000,B 0.000,C 180.000} C_DIS
LIN {X 99.002,Y 47.493,Z 70.173,A 180.000,B 0.000,C 180.000} C_DIS
LIN {X 98.503,Y 47.493,Z 70.228,A 180.000,B 0.000,C 180.000} C_DIS
LIN {X 97.903,Y 47.493,Z 70.247,A 180.000,B 0.000,C 180.000} C_DIS
LIN {X 95.136,Y 47.493,Z 70.247,A 180.000,B 0.000,C 180.000} C_DIS
LIN {X 95.136,Y 47.493,Z 72.155,A 180.000,B 0.000,C 180.000} C_DIS
LIN {X 89.827,Y 47.493,Z 74.364,A 180.000,B 0.000,C 180.000} C_DIS
LIN {X 84.548,Y 47.493,Z 74.361,A 180.000,B 0.000,C 180.000} C_DIS
LIN {X 83.778,Y 47.493,Z 73.716,A 180.000,B 0.000,C 180.000} C_DIS
LIN {X 83.050,Y 47.493,Z 73.150,A 180.000,B 0.000,C 180.000} C_DIS
LIN {X 82.293,Y 47.493,Z 72.608,A 180.000,B 0.000,C 180.000} C_DIS
LIN {X 81.607,Y 47.493,Z 72.158,A 180.000,B 0.000,C 180.000} C_DIS
LIN {X 80.939,Y 47.493,Z 71.761,A 180.000,B 0.000,C 180.000} C_DIS
LIN {X 80.285,Y 47.493,Z 71.411,A 180.000,B 0.000,C 180.000} C_DIS
LIN {X 79.637,Y 47.493,Z 71.102,A 180.000,B 0.000,C 180.000} C_DIS
LIN {X 79.019,Y 47.493,Z 70.844,A 180.000,B 0.000,C 180.000} C_DIS
LIN {X 78.399,Y 47.493,Z 70.622,A 180.000,B 0.000,C 180.000} C_DIS
LIN {X 77.777,Y 47.493,Z 70.435,A 180.000,B 0.000,C 180.000} C_DIS
LIN {X 77.695,Y 47.493,Z 70.415,A 180.000,B 0.000,C 180.000} C_DIS
LIN {X 77.273,Y 47.493,Z 70.531,A 180.000,B 0.000,C 180.000} C_DIS
LIN {X 76.649,Y 47.493,Z 70.735,A 180.000,B 0.000,C 180.000} C_DIS
LIN {X 76.021,Y 47.493,Z 70.978,A 180.000,B 0.000,C 180.000} C_DIS
LIN {X 75.389,Y 47.493,Z 71.257,A 180.000,B 0.000,C 180.000} C_DIS
LIN {X 74.767,Y 47.493,Z 71.565,A 180.000,B 0.000,C 180.000} C_DIS
LIN {X 74.141,Y 47.493,Z 71.907,A 180.000,B 0.000,C 180.000} C_DIS
LIN {X 73.514,Y 47.493,Z 72.279,A 180.000,B 0.000,C 180.000} C_DIS
LIN {X 72.874,Y 47.493,Z 72.687,A 180.000,B 0.000,C 180.000} C_DIS
LIN {X 72.195,Y 47.493,Z 73.149,A 180.000,B 0.000,C 180.000} C_DIS
LIN {X 71.297,Y 47.493,Z 73.798,A 180.000,B 0.000,C 180.000} C_DIS
LIN {X 70.468,Y 47.493,Z 74.436,A 180.000,B 0.000,C 180.000} C_DIS
LIN {X 69.326,Y 47.493,Z 75.345,A 180.000,B 0.000,C 180.000} C_DIS
LIN {X 66.108,Y 47.493,Z 77.983,A 180.000,B 0.000,C 180.000} C_DIS
LIN {X 64.949,Y 47.493,Z 78.895,A 180.000,B 0.000,C 180.000} C_DIS
LIN {X 64.333,Y 47.493,Z 79.359,A 180.000,B 0.000,C 180.000} C_DIS
LIN {X 63.769,Y 47.493,Z 79.770,A 180.000,B 0.000,C 180.000} C_DIS
LIN {X 63.193,Y 47.493,Z 80.171,A 180.000,B 0.000,C 180.000} C_DIS
LIN {X 62.608,Y 47.493,Z 80.558,A 180.000,B 0.000,C 180.000} C_DIS
LIN {X 62.014,Y 47.493,Z 80.929,A 180.000,B 0.000,C 180.000} C_DIS
LIN {X 61.413,Y 47.493,Z 81.279,A 180.000,B 0.000,C 180.000} C_DIS
LIN {X 60.764,Y 47.493,Z 81.624,A 180.000,B 0.000,C 180.000} C_DIS
LIN {X 60.127,Y 47.493,Z 81.925,A 180.000,B 0.000,C 180.000} C_DIS
LIN {X 59.460,Y 47.493,Z 82.198,A 180.000,B 0.000,C 180.000} C_DIS
LIN {X 58.761,Y 47.493,Z 82.440,A 180.000,B 0.000,C 180.000} C_DIS
LIN {X 58.023,Y 47.493,Z 82.651,A 180.000,B 0.000,C 180.000} C_DIS
LIN {X 57.229,Y 47.493,Z 82.829,A 180.000,B 0.000,C 180.000} C_DIS
LIN {X 56.354,Y 47.493,Z 82.971,A 180.000,B 0.000,C 180.000} C_DIS
LIN {X 55.765,Y 47.493,Z 83.038,A 180.000,B 0.000,C 180.000} C_DIS
LIN {X 55.203,Y 47.493,Z 83.083,A 180.000,B 0.000,C 180.000} C_DIS
LIN {X 54.585,Y 47.493,Z 83.114,A 180.000,B 0.000,C 180.000} C_DIS
LIN {X 53.803,Y 47.493,Z 83.130,A 180.000,B 0.000,C 180.000} C_DIS
LIN {X 53.493,Y 47.493,Z 83.119,A 180.000,B 0.000,C 180.000} C_DIS
LIN {X 53.420,Y 47.493,Z 83.103,A 180.000,B 0.000,C 180.000} C_DIS
LIN {X 53.416,Y 47.493,Z 62.000,A 180.000,B 0.000,C 180.000} C_DIS
LIN {X 38.972,Y 47.493,Z 62.000,A 180.000,B 0.000,C 180.000} C_DIS
LIN {X 38.972,Y 47.493,Z 57.000,A 180.000,B 0.000,C 180.000} C_DIS
LIN {X 8.770,Y 47.493,Z 57.000,A 180.000,B 0.000,C 180.000} C_DIS
LIN {X 8.770,Y 47.493,Z 52.000,A 180.000,B 0.000,C 180.000} C_DIS
LIN {X 2.500,Y 47.493,Z 52.000,A 180.000,B 0.000,C 180.000} C_DIS
LIN {X 2.500,Y 47.493,Z 45.000,A 180.000,B 0.000,C 180.000} C_DIS
LIN {X -0.010,Y 47.493,Z 45.000,A 180.000,B 0.000,C 180.000} C_DIS
; Link Move Starts
LIN {X -0.120,Y 47.493,Z 45.026,A 180.000,B 0.000,C 180.000} C_DIS
LIN {X -0.230,Y 47.493,Z 45.051,A 180.000,B 0.000,C 180.000} C_DIS
LIN {X -0.771,Y 47.805,Z 45.051,A 180.000,B 0.000,C 180.000} C_DIS
LIN {X -0.771,Y 48.430,Z 45.051,A 180.000,B 0.000,C 180.000} C_DIS
LIN {X -0.230,Y 48.743,Z 45.051,A 180.000,B 0.000,C 180.000} C_DIS
LIN {X -0.120,Y 48.743,Z 45.026,A 180.000,B 0.000,C 180.000} C_DIS
LIN {X -0.010,Y 48.743,Z 45.000,A 180.000,B 0.000,C 180.000} C_DIS
; Cutting Move Starts
LIN {X 2.500,Y 48.743,Z 45.000,A 180.000,B 0.000,C 180.000} C_DIS
LIN {X 2.500,Y 48.743,Z 52.000,A 180.000,B 0.000,C 180.000} C_DIS
LIN {X 8.236,Y 48.743,Z 52.000,A 180.000,B 0.000,C 180.000} C_DIS
LIN {X 8.236,Y 48.743,Z 57.000,A 180.000,B 0.000,C 180.000} C_DIS
LIN {X 37.722,Y 48.743,Z 57.000,A 180.000,B 0.000,C 180.000} C_DIS
LIN {X 37.722,Y 48.743,Z 62.000,A 180.000,B 0.000,C 180.000} C_DIS
LIN {X 49.711,Y 48.743,Z 62.000,A 180.000,B 0.000,C 180.000} C_DIS
LIN {X 49.711,Y 48.743,Z 82.728,A 180.000,B 0.000,C 180.000} C_DIS
LIN {X 49.720,Y 48.743,Z 82.766,A 180.000,B 0.000,C 180.000} C_DIS
LIN {X 49.771,Y 48.743,Z 82.828,A 180.000,B 0.000,C 180.000} C_DIS
LIN {X 49.877,Y 48.743,Z 82.900,A 180.000,B 0.000,C 180.000} C_DIS
LIN {X 50.016,Y 48.743,Z 82.965,A 180.000,B 0.000,C 180.000} C_DIS
LIN {X 50.195,Y 48.743,Z 83.025,A 180.000,B 0.000,C 180.000} C_DIS
LIN {X 50.410,Y 48.743,Z 83.077,A 180.000,B 0.000,C 180.000} C_DIS
LIN {X 50.704,Y 48.743,Z 83.123,A 180.000,B 0.000,C 180.000} C_DIS
LIN {X 51.036,Y 48.743,Z 83.146,A 180.000,B 0.000,C 180.000} C_DIS
LIN {X 55.438,Y 48.743,Z 83.148,A 180.000,B 0.000,C 180.000} C_DIS
LIN {X 55.880,Y 48.743,Z 83.135,A 180.000,B 0.000,C 180.000} C_DIS
LIN {X 56.394,Y 48.743,Z 83.100,A 180.000,B 0.000,C 180.000} C_DIS
LIN {X 56.895,Y 48.743,Z 83.043,A 180.000,B 0.000,C 180.000} C_DIS
LIN {X 57.360,Y 48.743,Z 82.970,A 180.000,B 0.000,C 180.000} C_DIS
LIN {X 58.043,Y 48.743,Z 82.825,A 180.000,B 0.000,C 180.000} C_DIS
LIN {X 58.699,Y 48.743,Z 82.645,A 180.000,B 0.000,C 180.000} C_DIS
LIN {X 59.343,Y 48.743,Z 82.432,A 180.000,B 0.000,C 180.000} C_DIS
LIN {X 59.979,Y 48.743,Z 82.186,A 180.000,B 0.000,C 180.000} C_DIS
LIN {X 60.607,Y 48.743,Z 81.911,A 180.000,B 0.000,C 180.000} C_DIS
LIN {X 61.221,Y 48.743,Z 81.609,A 180.000,B 0.000,C 180.000} C_DIS
LIN {X 61.835,Y 48.743,Z 81.279,A 180.000,B 0.000,C 180.000} C_DIS
LIN {X 62.435,Y 48.743,Z 80.929,A 180.000,B 0.000,C 180.000} C_DIS
LIN {X 63.029,Y 48.743,Z 80.558,A 180.000,B 0.000,C 180.000} C_DIS
LIN {X 63.614,Y 48.743,Z 80.171,A 180.000,B 0.000,C 180.000} C_DIS
LIN {X 64.191,Y 48.743,Z 79.770,A 180.000,B 0.000,C 180.000} C_DIS
LIN {X 64.755,Y 48.743,Z 79.359,A 180.000,B 0.000,C 180.000} C_DIS
LIN {X 65.371,Y 48.743,Z 78.895,A 180.000,B 0.000,C 180.000} C_DIS
LIN {X 66.530,Y 48.743,Z 77.983,A 180.000,B 0.000,C 180.000} C_DIS
LIN {X 69.748,Y 48.743,Z 75.345,A 180.000,B 0.000,C 180.000} C_DIS
LIN {X 70.890,Y 48.743,Z 74.436,A 180.000,B 0.000,C 180.000} C_DIS
LIN {X 71.719,Y 48.743,Z 73.798,A 180.000,B 0.000,C 180.000} C_DIS
LIN {X 72.617,Y 48.743,Z 73.149,A 180.000,B 0.000,C 180.000} C_DIS
LIN {X 73.296,Y 48.743,Z 72.687,A 180.000,B 0.000,C 180.000} C_DIS
LIN {X 73.935,Y 48.743,Z 72.279,A 180.000,B 0.000,C 180.000} C_DIS
LIN {X 74.563,Y 48.743,Z 71.907,A 180.000,B 0.000,C 180.000} C_DIS
LIN {X 75.188,Y 48.743,Z 71.566,A 180.000,B 0.000,C 180.000} C_DIS
LIN {X 75.810,Y 48.743,Z 71.257,A 180.000,B 0.000,C 180.000} C_DIS
LIN {X 76.442,Y 48.743,Z 70.978,A 180.000,B 0.000,C 180.000} C_DIS
LIN {X 77.071,Y 48.743,Z 70.735,A 180.000,B 0.000,C 180.000} C_DIS
LIN {X 77.694,Y 48.743,Z 70.531,A 180.000,B 0.000,C 180.000} C_DIS
LIN {X 78.115,Y 48.743,Z 70.415,A 180.000,B 0.000,C 180.000} C_DIS
LIN {X 78.197,Y 48.743,Z 70.435,A 180.000,B 0.000,C 180.000} C_DIS
LIN {X 78.820,Y 48.743,Z 70.622,A 180.000,B 0.000,C 180.000} C_DIS
LIN {X 79.440,Y 48.743,Z 70.843,A 180.000,B 0.000,C 180.000} C_DIS
LIN {X 80.058,Y 48.743,Z 71.101,A 180.000,B 0.000,C 180.000} C_DIS
LIN {X 80.707,Y 48.743,Z 71.411,A 180.000,B 0.000,C 180.000} C_DIS
LIN {X 81.361,Y 48.743,Z 71.760,A 180.000,B 0.000,C 180.000} C_DIS
LIN {X 82.028,Y 48.743,Z 72.157,A 180.000,B 0.000,C 180.000} C_DIS
LIN {X 82.714,Y 48.743,Z 72.607,A 180.000,B 0.000,C 180.000} C_DIS
LIN {X 83.471,Y 48.743,Z 73.150,A 180.000,B 0.000,C 180.000} C_DIS
LIN {X 84.200,Y 48.743,Z 73.716,A 180.000,B 0.000,C 180.000} C_DIS
LIN {X 84.969,Y 48.743,Z 74.361,A 180.000,B 0.000,C 180.000} C_DIS
LIN {X 90.247,Y 48.743,Z 74.364,A 180.000,B 0.000,C 180.000} C_DIS
LIN {X 95.558,Y 48.743,Z 72.155,A 180.000,B 0.000,C 180.000} C_DIS
LIN {X 95.558,Y 48.743,Z 70.247,A 180.000,B 0.000,C 180.000} C_DIS
LIN {X 97.772,Y 48.743,Z 70.247,A 180.000,B 0.000,C 180.000} C_DIS
LIN {X 98.387,Y 48.743,Z 70.227,A 180.000,B 0.000,C 180.000} C_DIS
LIN {X 98.894,Y 48.743,Z 70.172,A 180.000,B 0.000,C 180.000} C_DIS
LIN {X 99.404,Y 48.743,Z 70.079,A 180.000,B 0.000,C 180.000} C_DIS
LIN {X 99.942,Y 48.743,Z 69.940,A 180.000,B 0.000,C 180.000} C_DIS
LIN {X 100.437,Y 48.743,Z 69.770,A 180.000,B 0.000,C 180.000} C_DIS
LIN {X 100.922,Y 48.743,Z 69.562,A 180.000,B 0.000,C 180.000} C_DIS
LIN {X 101.388,Y 48.743,Z 69.321,A 180.000,B 0.000,C 180.000} C_DIS
LIN {X 101.835,Y 48.743,Z 69.045,A 180.000,B 0.000,C 180.000} C_DIS
LIN {X 102.261,Y 48.743,Z 68.737,A 180.000,B 0.000,C 180.000} C_DIS
LIN {X 102.645,Y 48.743,Z 68.412,A 180.000,B 0.000,C 180.000} C_DIS
LIN {X 103.022,Y 48.743,Z 68.044,A 180.000,B 0.000,C 180.000} C_DIS
LIN {X 103.369,Y 48.743,Z 67.650,A 180.000,B 0.000,C 180.000} C_DIS
LIN {X 103.684,Y 48.743,Z 67.231,A 180.000,B 0.000,C 180.000} C_DIS
LIN {X 103.979,Y 48.743,Z 66.771,A 180.000,B 0.000,C 180.000} C_DIS
LIN {X 104.227,Y 48.743,Z 66.307,A 180.000,B 0.000,C 180.000} C_DIS
LIN {X 104.439,Y 48.743,Z 65.827,A 180.000,B 0.000,C 180.000} C_DIS
LIN {X 104.614,Y 48.743,Z 65.335,A 180.000,B 0.000,C 180.000} C_DIS
LIN {X 104.746,Y 48.743,Z 64.852,A 180.000,B 0.000,C 180.000} C_DIS
LIN {X 104.849,Y 48.743,Z 64.329,A 180.000,B 0.000,C 180.000} C_DIS
LIN {X 104.910,Y 48.743,Z 63.814,A 180.000,B 0.000,C 180.000} C_DIS
LIN {X 104.933,Y 48.743,Z 63.296,A 180.000,B 0.000,C 180.000} C_DIS
LIN {X 104.935,Y 48.743,Z 62.000,A 180.000,B 0.000,C 180.000} C_DIS
LIN {X 117.278,Y 48.743,Z 62.000,A 180.000,B 0.000,C 180.000} C_DIS
LIN {X 117.278,Y 48.743,Z 57.000,A 180.000,B 0.000,C 180.000} C_DIS
LIN {X 146.761,Y 48.743,Z 57.000,A 180.000,B 0.000,C 180.000} C_DIS
LIN {X 146.764,Y 48.743,Z 52.000,A 180.000,B 0.000,C 180.000} C_DIS
LIN {X 152.500,Y 48.743,Z 52.000,A 180.000,B 0.000,C 180.000} C_DIS
LIN {X 152.500,Y 48.743,Z 45.000,A 180.000,B 0.000,C 180.000} C_DIS
LIN {X 155.010,Y 48.743,Z 45.000,A 180.000,B 0.000,C 180.000} C_DIS
; Link Move Starts
LIN {X 155.120,Y 48.743,Z 45.026,A 180.000,B 0.000,C 180.000} C_DIS
LIN {X 155.230,Y 48.743,Z 45.051,A 180.000,B 0.000,C 180.000} C_DIS
LIN {X 155.771,Y 49.055,Z 45.051,A 180.000,B 0.000,C 180.000} C_DIS
LIN {X 155.771,Y 49.680,Z 45.051,A 180.000,B 0.000,C 180.000} C_DIS
LIN {X 155.230,Y 49.993,Z 45.051,A 180.000,B 0.000,C 180.000} C_DIS
LIN {X 155.120,Y 49.993,Z 45.026,A 180.000,B 0.000,C 180.000} C_DIS
LIN {X 155.010,Y 49.993,Z 45.000,A 180.000,B 0.000,C 180.000} C_DIS
; Cutting Move Starts
